KUKA KRL program: ps_ltc_geo_c1_bolha.src, ps_ltc_geo_c1_bolha.dat

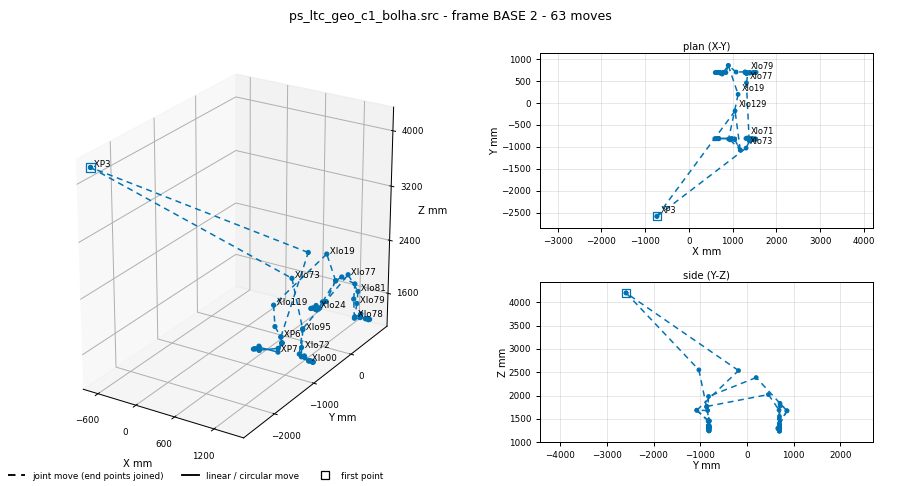
[picture p0: tool path of ps_ltc_geo_c1_bolha.src in frame BASE 2, 63 of 63 moves have a stored position in this frame; points joined in program order, loops and branches not executed]
--- ps_ltc_geo_c1_bolha.src ---
&ACCESS RVO1
&REL 30
&COMMENT SOLDA GEO C1 ACCELO
&PARAM DISKPATH = KRC:\R1\Program\SOLDA LTC
DEF ps_ltc_geo_c1_bolha( )
;FOLD INI
;FOLD SPOTTECH INI

;ENDFOLD (SPOTTECH INI)
;FOLD GRIPPERTECH INI
USER_GRP(0,DUMMY,DUMMY,GDEFAULT)
;ENDFOLD (GRIPPERTECH INI)
  ;FOLD USER INI
    ;Make your modifications here

  ;ENDFOLD (USER INI)
;ENDFOLD (INI)

; Caracterização dos meios de produção:
; Versão Atual:
; 15/07/2013 12:00 Name: P13.050-R5 CHANGES: Solda Geometria Accelo
; C1

chk_w1_wechs_ok ( )      ; CHECK FERRAMENTA: C1

;FOLD PTP P3 CONT Vel=100 % PDAT34 Tool[1]:Gun C1 Base[2]:ACCELO;%{PE}%R 8.2.20,%MKUKATPBASIS,%CMOVE,%VPTP,%P 1:PTP, 2:P3, 3:C_DIS, 5:100, 7:PDAT34
$BWDSTART=FALSE
PDAT_ACT=PPDAT34
FDAT_ACT=FP3
BAS(#PTP_PARAMS,100)
PTP XP3 C_DIS
;ENDFOLD

if MaxStandMenge (1) then
 MaxStandmengeErreicht (1)
endif

IF (NOT(GHOST())) THEN
if Elektrodenwechsel (1) then
 e_fraes1 ()
endif
ENDIF
;FOLD  ;%{PE}%R 8.2.20,%MKUKATPBASIS,%CCOMMENT,%VNORMAL,%P 2:
;ENDFOLD
;FOLD OUT 3339 'R5 aguarda lib soldar geometria' State=TRUE ;%{PE}%R 8.2.20,%MKUKATPBASIS,%COUT,%VOUTX,%P 2:3339, 3:R5 aguarda lib soldar geometria, 5:TRUE, 6:
$OUT[3339]=TRUE
;ENDFOLD
;FOLD WAIT FOR ( IN 3339 'Aguarda lib soldar geometria' );%{PE}%R 8.2.20,%MKUKATPBASIS,%CEXT_WAIT_FOR,%VEXT_WAIT_FOR,%P 2:, 4:, 5:$IN, 6:3339, 7:Aguarda lib soldar geometria, 9:
WAIT FOR  ( $IN[3339] )
;ENDFOLD
;FOLD OUT 3339 'R5 aguarda lib soldar geometria' State=FALSE ;%{PE}%R 8.2.20,%MKUKATPBASIS,%COUT,%VOUTX,%P 2:3339, 3:R5 aguarda lib soldar geometria, 5:FALSE, 6:
$OUT[3339]=FALSE
;ENDFOLD
;FOLD OUT 3344 'R5 entregou peca geo' State=FALSE ;%{PE}%R 8.2.20,%MKUKATPBASIS,%COUT,%VOUTX,%P 2:3344, 3:R5 entregou peca geo, 5:FALSE, 6:
$OUT[3344]=FALSE
;ENDFOLD

;FOLD PTP lo73 CONT Vel=100 % P_OLP1 Tool[1]:Gun C1 Base[2]:ACCELO;%{PE}%R 8.2.20,%MKUKATPBASIS,%CMOVE,%VPTP,%P 1:PTP, 2:lo73, 3:C_DIS, 5:100, 7:P_OLP1
$BWDSTART=FALSE
PDAT_ACT=PP_OLP1
FDAT_ACT=Flo73
BAS(#PTP_PARAMS,100)
PTP Xlo73 C_DIS
;ENDFOLD


;aqui
;FOLD PTP lo95 CONT Vel=100 % P_OLP10 Tool[1]:Gun C1 Base[2]:ACCELO;%{PE}%R8.2,%MKUKATPBASIS,%CMOVE,%VPTP,%P 1:PTP, 2:lo95, 3:C_DIS, 5:100, 7:P_OLP10
$BWDSTART = FALSE
PDAT_ACT= PP_OLP10
FDAT_ACT= Flo95
BAS(#PTP_PARAMS,100)
PTP Xlo95 C_DIS
;ENDFOLD
;FOLD PTP lo72 CONT Vel=100 % P_OLP11 Tool[1]:Gun C1 Base[2]:ACCELO;%{PE}%R8.2,%MKUKATPBASIS,%CMOVE,%VPTP,%P 1:PTP, 2:lo72, 3:C_DIS, 5:100, 7:P_OLP11
$BWDSTART = FALSE
PDAT_ACT= PP_OLP11
FDAT_ACT= Flo72
BAS(#PTP_PARAMS,100)
PTP Xlo72 C_DIS
;ENDFOLD


;FOLD PTP lo71 CONT Vel=100 % P_OLP12 Tool[1]:Gun C1 Base[2]:ACCELO;%{PE}%R8.2,%MKUKATPBASIS,%CMOVE,%VPTP,%P 1:PTP, 2:lo71, 3:C_DIS, 5:100, 7:P_OLP12
$BWDSTART = FALSE
PDAT_ACT= PP_OLP12
FDAT_ACT= Flo71
BAS(#PTP_PARAMS,100)
PTP Xlo71 C_DIS
;ENDFOLD
;FOLD PTP lo00 CONT Vel=100 % PDAT1 Tool[1]:Gun C1 Base[2]:ACCELO;%{PE}%R 8.2.20,%MKUKATPBASIS,%CMOVE,%VPTP,%P 1:PTP, 2:lo00, 3:C_DIS, 5:100, 7:PDAT1
$BWDSTART=FALSE
PDAT_ACT=PPDAT1
FDAT_ACT=Flo00
BAS(#PTP_PARAMS,100)
PTP Xlo00 C_DIS
;ENDFOLD
;FOLD PTP lo01 CONT Vel=100 % PDAT2 Tool[1]:Gun C1 Base[2]:ACCELO;%{PE}%R 8.2.20,%MKUKATPBASIS,%CMOVE,%VPTP,%P 1:PTP, 2:lo01, 3:C_DIS, 5:100, 7:PDAT2
$BWDSTART=FALSE
PDAT_ACT=PPDAT2
FDAT_ACT=Flo01
BAS(#PTP_PARAMS,100)
PTP Xlo01 C_DIS
;ENDFOLD

;FOLD ; swp_60_0421;%{PE}%R 8.2.20,%MKUKATPBASIS,%CCOMMENT,%VNORMAL,%P 2:swp_60_0421
;ENDFOLD
;FOLD PTP lpt_60_0421 P_OLP13 SPOT Gun=1 RETR CLS PgNo1=2 ACTIVE=1 Tool[1]:Gun C1 Base[2]:ACCELO;%{PE}%R 8.2.2,%MKUKATPSPOT,%CSPOT,%VPTP,%P 1:PTP, 2:lpt_60_0421, 3:, 5:100, 7:P_OLP13, 10:1, 12:#FIRST, 14:#CLO, 16:2, 18:1, 20:1, 22:0, 24:1, 25:S_OLP2
$BWDSTART=FALSE
PDAT_ACT=PP_OLP13
FDAT_ACT=Flpt_60_0421
BAS(#PTP_PARAMS,PP_OLP13.VEL)
S_ACT.GUN=1
S_ACT.PAIR=SDEFAULT.PAIR
S_ACT.RETR=#CLO
S_ACT.CLO_TM=1
S_ACT.PGNO1=2
S_ACT.PGNO2=SDEFAULT.PGNO2
S_ACT.PRESS1=SDEFAULT.PRESS1
S_ACT.PRESS2=SDEFAULT.PRESS2
S_READY=FALSE
PTP Xlpt_60_0421
USERSPOT(#SPOT, S_ACT)
WAIT FOR S_READY
;ENDFOLD

;FOLD ; swp_60_0419;%{PE}%R 8.2.20,%MKUKATPBASIS,%CCOMMENT,%VNORMAL,%P 2:swp_60_0419
;ENDFOLD
;FOLD PTP lpt_60_0419 P_OLP14 SPOT Gun=1 RETR CLS PgNo1=3 ACTIVE=1 Tool[1]:Gun C1 Base[2]:ACCELO;%{PE}%R 8.2.2,%MKUKATPSPOT,%CSPOT,%VPTP,%P 1:PTP, 2:lpt_60_0419, 3:, 5:100, 7:P_OLP14, 10:1, 12:#FIRST, 14:#CLO, 16:3, 18:1, 20:1, 22:0, 24:1, 25:S_OLP3
$BWDSTART=FALSE
PDAT_ACT=PP_OLP14
FDAT_ACT=Flpt_60_0419
BAS(#PTP_PARAMS,PP_OLP14.VEL)
S_ACT.GUN=1
S_ACT.PAIR=SDEFAULT.PAIR
S_ACT.RETR=#CLO
S_ACT.CLO_TM=1
S_ACT.PGNO1=3
S_ACT.PGNO2=SDEFAULT.PGNO2
S_ACT.PRESS1=SDEFAULT.PRESS1
S_ACT.PRESS2=SDEFAULT.PRESS2
S_READY=FALSE
PTP Xlpt_60_0419
USERSPOT(#SPOT, S_ACT)
WAIT FOR S_READY
;ENDFOLD

;FOLD ; swp_60_0417;%{PE}%R 8.2.20,%MKUKATPBASIS,%CCOMMENT,%VNORMAL,%P 2:swp_60_0417
;ENDFOLD
;FOLD PTP lpt_60_0417 P_OLP15 SPOT Gun=1 RETR CLS PgNo1=4 ACTIVE=1 Tool[1]:Gun C1 Base[2]:ACCELO;%{PE}%R 8.2.2,%MKUKATPSPOT,%CSPOT,%VPTP,%P 1:PTP, 2:lpt_60_0417, 3:, 5:100, 7:P_OLP15, 10:1, 12:#FIRST, 14:#CLO, 16:4, 18:1, 20:1, 22:0, 24:1, 25:S_OLP4
$BWDSTART=FALSE
PDAT_ACT=PP_OLP15
FDAT_ACT=Flpt_60_0417
BAS(#PTP_PARAMS,PP_OLP15.VEL)
S_ACT.GUN=1
S_ACT.PAIR=SDEFAULT.PAIR
S_ACT.RETR=#CLO
S_ACT.CLO_TM=1
S_ACT.PGNO1=4
S_ACT.PGNO2=SDEFAULT.PGNO2
S_ACT.PRESS1=SDEFAULT.PRESS1
S_ACT.PRESS2=SDEFAULT.PRESS2
S_READY=FALSE
PTP Xlpt_60_0417
USERSPOT(#SPOT, S_ACT)
WAIT FOR S_READY
;ENDFOLD

;FOLD ; swp_60_0415;%{PE}%R 8.2.20,%MKUKATPBASIS,%CCOMMENT,%VNORMAL,%P 2:swp_60_0415
;ENDFOLD
;FOLD PTP lpt_60_0415 P_OLP16 SPOT Gun=1 RETR OPN PgNo1=5 ACTIVE=1 Tool[1]:Gun C1 Base[2]:ACCELO;%{PE}%R 8.2.2,%MKUKATPSPOT,%CSPOT,%VPTP,%P 1:PTP, 2:lpt_60_0415, 3:, 5:100, 7:P_OLP16, 10:1, 12:#FIRST, 14:#OPN, 16:5, 18:1, 20:1, 22:0, 24:1, 25:S_OLP5
$BWDSTART=FALSE
PDAT_ACT=PP_OLP16
FDAT_ACT=Flpt_60_0415
BAS(#PTP_PARAMS,PP_OLP16.VEL)
S_ACT.GUN=1
S_ACT.PAIR=SDEFAULT.PAIR
S_ACT.RETR=#OPN
S_ACT.CLO_TM=1
S_ACT.PGNO1=5
S_ACT.PGNO2=SDEFAULT.PGNO2
S_ACT.PRESS1=SDEFAULT.PRESS1
S_ACT.PRESS2=SDEFAULT.PRESS2
S_READY=FALSE
PTP Xlpt_60_0415
USERSPOT(#SPOT, S_ACT)
WAIT FOR S_READY
;ENDFOLD

;FOLD PTP lo75 CONT Vel=100 % P_OLP17 Tool[1]:Gun C1 Base[2]:ACCELO;%{PE}%R8.2,%MKUKATPBASIS,%CMOVE,%VPTP,%P 1:PTP, 2:lo75, 3:C_DIS, 5:100, 7:P_OLP17
$BWDSTART = FALSE
PDAT_ACT= PP_OLP17
FDAT_ACT= Flo75
BAS(#PTP_PARAMS,100)
PTP Xlo75 C_DIS
;ENDFOLD

;FOLD ; swp_60_0413;%{PE}%R 8.2.20,%MKUKATPBASIS,%CCOMMENT,%VNORMAL,%P 2:swp_60_0413
;ENDFOLD
;FOLD PTP lpt_60_0413 P_OLP18 SPOT Gun=1 RETR OPN PgNo1=6 ACTIVE=1 Tool[1]:Gun C1 Base[2]:ACCELO;%{PE}%R 8.2.2,%MKUKATPSPOT,%CSPOT,%VPTP,%P 1:PTP, 2:lpt_60_0413, 3:, 5:100, 7:P_OLP18, 10:1, 12:#FIRST, 14:#OPN, 16:6, 18:1, 20:1, 22:0, 24:1, 25:S_OLP6
$BWDSTART=FALSE
PDAT_ACT=PP_OLP18
FDAT_ACT=Flpt_60_0413
BAS(#PTP_PARAMS,PP_OLP18.VEL)
S_ACT.GUN=1
S_ACT.PAIR=SDEFAULT.PAIR
S_ACT.RETR=#OPN
S_ACT.CLO_TM=1
S_ACT.PGNO1=6
S_ACT.PGNO2=SDEFAULT.PGNO2
S_ACT.PRESS1=SDEFAULT.PRESS1
S_ACT.PRESS2=SDEFAULT.PRESS2
S_READY=FALSE
PTP Xlpt_60_0413
USERSPOT(#SPOT, S_ACT)
WAIT FOR S_READY
;ENDFOLD

;FOLD PTP lo76 CONT Vel=100 % P_OLP19 Tool[1]:Gun C1 Base[2]:ACCELO;%{PE}%R8.2,%MKUKATPBASIS,%CMOVE,%VPTP,%P 1:PTP, 2:lo76, 3:C_DIS, 5:100, 7:P_OLP19
$BWDSTART = FALSE
PDAT_ACT= PP_OLP19
FDAT_ACT= Flo76
BAS(#PTP_PARAMS,100)
PTP Xlo76 C_DIS
;ENDFOLD
;FOLD PTP lo80 CONT Vel=100 % P_OLP20 Tool[1]:Gun C1 Base[2]:ACCELO;%{PE}%R8.2,%MKUKATPBASIS,%CMOVE,%VPTP,%P 1:PTP, 2:lo80, 3:C_DIS, 5:100, 7:P_OLP20
$BWDSTART = FALSE
PDAT_ACT= PP_OLP20
FDAT_ACT= Flo80
BAS(#PTP_PARAMS,100)
PTP Xlo80 C_DIS
;ENDFOLD
;FOLD PTP lo77 CONT Vel=100 % P_OLP21 Tool[1]:Gun C1 Base[2]:ACCELO;%{PE}%R8.2,%MKUKATPBASIS,%CMOVE,%VPTP,%P 1:PTP, 2:lo77, 3:C_DIS, 5:100, 7:P_OLP21
$BWDSTART = FALSE
PDAT_ACT= PP_OLP21
FDAT_ACT= Flo77
BAS(#PTP_PARAMS,100)
PTP Xlo77 C_DIS
;ENDFOLD
;FOLD PTP lo81 CONT Vel=100 % P_OLP22 Tool[1]:Gun C1 Base[2]:ACCELO;%{PE}%R8.2,%MKUKATPBASIS,%CMOVE,%VPTP,%P 1:PTP, 2:lo81, 3:C_DIS, 5:100, 7:P_OLP22
$BWDSTART = FALSE
PDAT_ACT= PP_OLP22
FDAT_ACT= Flo81
BAS(#PTP_PARAMS,100)
PTP Xlo81 C_DIS
;ENDFOLD
;FOLD PTP lo79 CONT Vel=100 % P_OLP23 Tool[1]:Gun C1 Base[2]:ACCELO;%{PE}%R8.2,%MKUKATPBASIS,%CMOVE,%VPTP,%P 1:PTP, 2:lo79, 3:C_DIS, 5:100, 7:P_OLP23
$BWDSTART = FALSE
PDAT_ACT= PP_OLP23
FDAT_ACT= Flo79
BAS(#PTP_PARAMS,100)
PTP Xlo79 C_DIS
;ENDFOLD
;FOLD PTP lo78 CONT Vel=100 % P_OLP24 Tool[1]:Gun C1 Base[2]:ACCELO;%{PE}%R8.2,%MKUKATPBASIS,%CMOVE,%VPTP,%P 1:PTP, 2:lo78, 3:C_DIS, 5:100, 7:P_OLP24
$BWDSTART = FALSE
PDAT_ACT= PP_OLP24
FDAT_ACT= Flo78
BAS(#PTP_PARAMS,100)
PTP Xlo78 C_DIS
;ENDFOLD
;FOLD PTP lo03 CONT Vel=100 % PDAT4 Tool[1]:Gun C1 Base[2]:ACCELO;%{PE}%R 8.2.20,%MKUKATPBASIS,%CMOVE,%VPTP,%P 1:PTP, 2:lo03, 3:C_DIS, 5:100, 7:PDAT4
$BWDSTART=FALSE
PDAT_ACT=PPDAT4
FDAT_ACT=Flo03
BAS(#PTP_PARAMS,100)
PTP Xlo03 C_DIS
;ENDFOLD

;FOLD ; swp_60_0414;%{PE}%R 8.2.20,%MKUKATPBASIS,%CCOMMENT,%VNORMAL,%P 2:swp_60_0414
;ENDFOLD
;FOLD PTP lpt_60_0414 P_OLP25 SPOT Gun=1 RETR OPN PgNo1=7 ACTIVE=1 Tool[1]:Gun C1 Base[2]:ACCELO;%{PE}%R 8.2.2,%MKUKATPSPOT,%CSPOT,%VPTP,%P 1:PTP, 2:lpt_60_0414, 3:, 5:100, 7:P_OLP25, 10:1, 12:#FIRST, 14:#OPN, 16:7, 18:1, 20:1, 22:0, 24:1, 25:S_OLP7
$BWDSTART=FALSE
PDAT_ACT=PP_OLP25
FDAT_ACT=Flpt_60_0414
BAS(#PTP_PARAMS,PP_OLP25.VEL)
S_ACT.GUN=1
S_ACT.PAIR=SDEFAULT.PAIR
S_ACT.RETR=#OPN
S_ACT.CLO_TM=1
S_ACT.PGNO1=7
S_ACT.PGNO2=SDEFAULT.PGNO2
S_ACT.PRESS1=SDEFAULT.PRESS1
S_ACT.PRESS2=SDEFAULT.PRESS2
S_READY=FALSE
PTP Xlpt_60_0414
USERSPOT(#SPOT, S_ACT)
WAIT FOR S_READY
;ENDFOLD

;FOLD PTP lo82 CONT Vel=100 % P_OLP26 Tool[1]:Gun C1 Base[2]:ACCELO;%{PE}%R8.2,%MKUKATPBASIS,%CMOVE,%VPTP,%P 1:PTP, 2:lo82, 3:C_DIS, 5:100, 7:P_OLP26
$BWDSTART = FALSE
PDAT_ACT= PP_OLP26
FDAT_ACT= Flo82
BAS(#PTP_PARAMS,100)
PTP Xlo82 C_DIS
;ENDFOLD

;FOLD ; swp_60_0416;%{PE}%R 8.2.20,%MKUKATPBASIS,%CCOMMENT,%VNORMAL,%P 2:swp_60_0416
;ENDFOLD
;FOLD PTP lpt_60_0416 P_OLP27 SPOT Gun=1 RETR CLS PgNo1=8 ACTIVE=1 Tool[1]:Gun C1 Base[2]:ACCELO;%{PE}%R 8.2.2,%MKUKATPSPOT,%CSPOT,%VPTP,%P 1:PTP, 2:lpt_60_0416, 3:, 5:100, 7:P_OLP27, 10:1, 12:#FIRST, 14:#CLO, 16:8, 18:1, 20:1, 22:0, 24:1, 25:S_OLP8
$BWDSTART=FALSE
PDAT_ACT=PP_OLP27
FDAT_ACT=Flpt_60_0416
BAS(#PTP_PARAMS,PP_OLP27.VEL)
S_ACT.GUN=1
S_ACT.PAIR=SDEFAULT.PAIR
S_ACT.RETR=#CLO
S_ACT.CLO_TM=1
S_ACT.PGNO1=8
S_ACT.PGNO2=SDEFAULT.PGNO2
S_ACT.PRESS1=SDEFAULT.PRESS1
S_ACT.PRESS2=SDEFAULT.PRESS2
S_READY=FALSE
PTP Xlpt_60_0416
USERSPOT(#SPOT, S_ACT)
WAIT FOR S_READY
;ENDFOLD

;FOLD ; swp_60_0418;%{PE}%R 8.2.20,%MKUKATPBASIS,%CCOMMENT,%VNORMAL,%P 2:swp_60_0418
;ENDFOLD
;FOLD PTP lpt_60_0418 P_OLP28 SPOT Gun=1 RETR CLS PgNo1=9 ACTIVE=1 Tool[1]:Gun C1 Base[2]:ACCELO;%{PE}%R 8.2.2,%MKUKATPSPOT,%CSPOT,%VPTP,%P 1:PTP, 2:lpt_60_0418, 3:, 5:100, 7:P_OLP28, 10:1, 12:#FIRST, 14:#CLO, 16:9, 18:1, 20:1, 22:0, 24:1, 25:S_OLP9
$BWDSTART=FALSE
PDAT_ACT=PP_OLP28
FDAT_ACT=Flpt_60_0418
BAS(#PTP_PARAMS,PP_OLP28.VEL)
S_ACT.GUN=1
S_ACT.PAIR=SDEFAULT.PAIR
S_ACT.RETR=#CLO
S_ACT.CLO_TM=1
S_ACT.PGNO1=9
S_ACT.PGNO2=SDEFAULT.PGNO2
S_ACT.PRESS1=SDEFAULT.PRESS1
S_ACT.PRESS2=SDEFAULT.PRESS2
S_READY=FALSE
PTP Xlpt_60_0418
USERSPOT(#SPOT, S_ACT)
WAIT FOR S_READY
;ENDFOLD

;FOLD ; swp_60_0420;%{PE}%R 8.2.20,%MKUKATPBASIS,%CCOMMENT,%VNORMAL,%P 2:swp_60_0420
;ENDFOLD
;FOLD PTP lpt_60_0420 P_OLP29 SPOT Gun=1 RETR CLS PgNo1=10 ACTIVE=1 Tool[1]:Gun C1 Base[2]:ACCELO;%{PE}%R 8.2.2,%MKUKATPSPOT,%CSPOT,%VPTP,%P 1:PTP, 2:lpt_60_0420, 3:, 5:100, 7:P_OLP29, 10:1, 12:#FIRST, 14:#CLO, 16:10, 18:1, 20:1, 22:0, 24:1, 25:S_OLP10
$BWDSTART=FALSE
PDAT_ACT=PP_OLP29
FDAT_ACT=Flpt_60_0420
BAS(#PTP_PARAMS,PP_OLP29.VEL)
S_ACT.GUN=1
S_ACT.PAIR=SDEFAULT.PAIR
S_ACT.RETR=#CLO
S_ACT.CLO_TM=1
S_ACT.PGNO1=10
S_ACT.PGNO2=SDEFAULT.PGNO2
S_ACT.PRESS1=SDEFAULT.PRESS1
S_ACT.PRESS2=SDEFAULT.PRESS2
S_READY=FALSE
PTP Xlpt_60_0420
USERSPOT(#SPOT, S_ACT)
WAIT FOR S_READY
;ENDFOLD

;FOLD PTP lo04 CONT Vel=100 % PDAT5 Tool[1]:Gun C1 Base[2]:ACCELO;%{PE}%R 8.2.20,%MKUKATPBASIS,%CMOVE,%VPTP,%P 1:PTP, 2:lo04, 3:C_DIS, 5:100, 7:PDAT5
$BWDSTART=FALSE
PDAT_ACT=PPDAT5
FDAT_ACT=Flo04
BAS(#PTP_PARAMS,100)
PTP Xlo04 C_DIS
;ENDFOLD

;FOLD ; swp_60_0422;%{PE}%R 8.2.20,%MKUKATPBASIS,%CCOMMENT,%VNORMAL,%P 2:swp_60_0422
;ENDFOLD
;FOLD PTP lpt_60_0422 P_OLP30 SPOT Gun=1 RETR OPN PgNo1=11 ACTIVE=1 Tool[1]:Gun C1 Base[2]:ACCELO;%{PE}%R 8.2.2,%MKUKATPSPOT,%CSPOT,%VPTP,%P 1:PTP, 2:lpt_60_0422, 3:, 5:100, 7:P_OLP30, 10:1, 12:#FIRST, 14:#OPN, 16:11, 18:1, 20:1, 22:0, 24:1, 25:S_OLP11
$BWDSTART=FALSE
PDAT_ACT=PP_OLP30
FDAT_ACT=Flpt_60_0422
BAS(#PTP_PARAMS,PP_OLP30.VEL)
S_ACT.GUN=1
S_ACT.PAIR=SDEFAULT.PAIR
S_ACT.RETR=#OPN
S_ACT.CLO_TM=1
S_ACT.PGNO1=11
S_ACT.PGNO2=SDEFAULT.PGNO2
S_ACT.PRESS1=SDEFAULT.PRESS1
S_ACT.PRESS2=SDEFAULT.PRESS2
S_READY=FALSE
PTP Xlpt_60_0422
USERSPOT(#SPOT, S_ACT)
WAIT FOR S_READY
;ENDFOLD

;FOLD PTP lo83 CONT Vel=100 % P_OLP31 Tool[1]:Gun C1 Base[2]:ACCELO;%{PE}%R8.2,%MKUKATPBASIS,%CMOVE,%VPTP,%P 1:PTP, 2:lo83, 3:C_DIS, 5:100, 7:P_OLP31
$BWDSTART = FALSE
PDAT_ACT= PP_OLP31
FDAT_ACT= Flo83
BAS(#PTP_PARAMS,100)
PTP Xlo83 C_DIS
;ENDFOLD
;FOLD PTP lo20 CONT Vel=100 % PDAT18 Tool[1]:Gun C1 Base[2]:ACCELO;%{PE}%R 8.2.20,%MKUKATPBASIS,%CMOVE,%VPTP,%P 1:PTP, 2:lo20, 3:C_DIS, 5:100, 7:PDAT18
$BWDSTART=FALSE
PDAT_ACT=PPDAT18
FDAT_ACT=Flo20
BAS(#PTP_PARAMS,100)
PTP Xlo20 C_DIS
;ENDFOLD
;FOLD PTP lo84 CONT Vel=100 % P_OLP32 Tool[1]:Gun C1 Base[2]:ACCELO;%{PE}%R8.2,%MKUKATPBASIS,%CMOVE,%VPTP,%P 1:PTP, 2:lo84, 3:C_DIS, 5:100, 7:P_OLP32
$BWDSTART = FALSE
PDAT_ACT= PP_OLP32
FDAT_ACT= Flo84
BAS(#PTP_PARAMS,100)
PTP Xlo84 C_DIS
;ENDFOLD
;FOLD PTP lo112 CONT Vel=100 % P_OLP53 Tool[1]:Gun C1 Base[2]:ACCELO;%{PE}%R8.2,%MKUKATPBASIS,%CMOVE,%VPTP,%P 1:PTP, 2:lo112, 3:C_DIS, 5:100, 7:P_OLP53
$BWDSTART = FALSE
PDAT_ACT= PP_OLP53
FDAT_ACT= Flo112
BAS(#PTP_PARAMS,100)
PTP Xlo112 C_DIS
;ENDFOLD
;FOLD PTP lo22 CONT Vel=100 % PDAT25 Tool[1]:Gun C1 Base[2]:ACCELO;%{PE}%R 8.2.20,%MKUKATPBASIS,%CMOVE,%VPTP,%P 1:PTP, 2:lo22, 3:C_DIS, 5:100, 7:PDAT25
$BWDSTART=FALSE
PDAT_ACT=PPDAT25
FDAT_ACT=Flo22
BAS(#PTP_PARAMS,100)
PTP Xlo22 C_DIS
;ENDFOLD
;FOLD PTP lo16 CONT Vel=100 % PDAT15 Tool[1]:Gun C1 Base[2]:ACCELO;%{PE}%R 8.2.20,%MKUKATPBASIS,%CMOVE,%VPTP,%P 1:PTP, 2:lo16, 3:C_DIS, 5:100, 7:PDAT15
$BWDSTART=FALSE
PDAT_ACT=PPDAT15
FDAT_ACT=Flo16
BAS(#PTP_PARAMS,100)
PTP Xlo16 C_DIS
;ENDFOLD
;FOLD PTP lo111 CONT Vel=100 % PDAT21 Tool[1]:Gun C1 Base[2]:ACCELO;%{PE}%R 8.2.20,%MKUKATPBASIS,%CMOVE,%VPTP,%P 1:PTP, 2:lo111, 3:C_DIS, 5:100, 7:PDAT21
$BWDSTART=FALSE
PDAT_ACT=PPDAT21
FDAT_ACT=Flo111
BAS(#PTP_PARAMS,100)
PTP Xlo111 C_DIS
;ENDFOLD
;FOLD PTP lo24 CONT Vel=100 % PDAT28 Tool[1]:Gun C1 Base[2]:ACCELO;%{PE}%R 8.2.20,%MKUKATPBASIS,%CMOVE,%VPTP,%P 1:PTP, 2:lo24, 3:C_DIS, 5:100, 7:PDAT28
$BWDSTART=FALSE
PDAT_ACT=PPDAT28
FDAT_ACT=Flo24
BAS(#PTP_PARAMS,100)
PTP Xlo24 C_DIS
;ENDFOLD

;FOLD ; swp_60_0412;%{PE}%R 8.2.20,%MKUKATPBASIS,%CCOMMENT,%VNORMAL,%P 2:swp_60_0412
;ENDFOLD
;FOLD PTP lpt_60_0412 PDAT27 SPOT Gun=1 RETR OPN PgNo1=15 ACTIVE=1 Tool[1]:Gun C1 Base[2]:ACCELO;%{PE}%R 8.2.2,%MKUKATPSPOT,%CSPOT,%VPTP,%P 1:PTP, 2:lpt_60_0412, 3:, 5:100, 7:PDAT27, 10:1, 12:#FIRST, 14:#OPN, 16:15, 18:1, 20:1, 22:0, 24:1, 25:S_OLP15
$BWDSTART=FALSE
PDAT_ACT=PPDAT27
FDAT_ACT=Flpt_60_0412
BAS(#PTP_PARAMS,PPDAT27.VEL)
S_ACT.GUN=1
S_ACT.PAIR=SDEFAULT.PAIR
S_ACT.RETR=#OPN
S_ACT.CLO_TM=1
S_ACT.PGNO1=15
S_ACT.PGNO2=SDEFAULT.PGNO2
S_ACT.PRESS1=SDEFAULT.PRESS1
S_ACT.PRESS2=SDEFAULT.PRESS2
S_READY=FALSE
PTP Xlpt_60_0412
USERSPOT(#SPOT, S_ACT)
WAIT FOR S_READY
;ENDFOLD

;FOLD PTP lo114 CONT Vel=100 % P_OLP58 Tool[1]:Gun C1 Base[2]:ACCELO;%{PE}%R8.2,%MKUKATPBASIS,%CMOVE,%VPTP,%P 1:PTP, 2:lo114, 3:C_DIS, 5:100, 7:P_OLP58
$BWDSTART = FALSE
PDAT_ACT= PP_OLP58
FDAT_ACT= Flo114
BAS(#PTP_PARAMS,100)
PTP Xlo114 C_DIS
;ENDFOLD

;FOLD ; swp_60_0410;%{PE}%R 8.2.20,%MKUKATPBASIS,%CCOMMENT,%VNORMAL,%P 2:swp_60_0410
;ENDFOLD
;FOLD PTP lpt_60_0410 PDAT29 SPOT Gun=1 RETR CLS PgNo1=16 ACTIVE=1 Tool[1]:Gun C1 Base[2]:ACCELO;%{PE}%R 8.2.2,%MKUKATPSPOT,%CSPOT,%VPTP,%P 1:PTP, 2:lpt_60_0410, 3:, 5:100, 7:PDAT29, 10:1, 12:#FIRST, 14:#CLO, 16:16, 18:1, 20:1, 22:0, 24:1, 25:S_OLP16
$BWDSTART=FALSE
PDAT_ACT=PPDAT29
FDAT_ACT=Flpt_60_0410
BAS(#PTP_PARAMS,PPDAT29.VEL)
S_ACT.GUN=1
S_ACT.PAIR=SDEFAULT.PAIR
S_ACT.RETR=#CLO
S_ACT.CLO_TM=1
S_ACT.PGNO1=16
S_ACT.PGNO2=SDEFAULT.PGNO2
S_ACT.PRESS1=SDEFAULT.PRESS1
S_ACT.PRESS2=SDEFAULT.PRESS2
S_READY=FALSE
PTP Xlpt_60_0410
USERSPOT(#SPOT, S_ACT)
WAIT FOR S_READY
;ENDFOLD

;FOLD ; swp_60_0408;%{PE}%R 8.2.20,%MKUKATPBASIS,%CCOMMENT,%VNORMAL,%P 2:swp_60_0408
;ENDFOLD
;FOLD PTP lpt_60_0408 P_OLP60 SPOT Gun=1 RETR CLS PgNo1=17 ACTIVE=1 Tool[1]:Gun C1 Base[2]:ACCELO;%{PE}%R 8.2.2,%MKUKATPSPOT,%CSPOT,%VPTP,%P 1:PTP, 2:lpt_60_0408, 3:, 5:100, 7:P_OLP60, 10:1, 12:#FIRST, 14:#CLO, 16:17, 18:1, 20:1, 22:0, 24:1, 25:S_OLP17
$BWDSTART=FALSE
PDAT_ACT=PP_OLP60
FDAT_ACT=Flpt_60_0408
BAS(#PTP_PARAMS,PP_OLP60.VEL)
S_ACT.GUN=1
S_ACT.PAIR=SDEFAULT.PAIR
S_ACT.RETR=#CLO
S_ACT.CLO_TM=1
S_ACT.PGNO1=17
S_ACT.PGNO2=SDEFAULT.PGNO2
S_ACT.PRESS1=SDEFAULT.PRESS1
S_ACT.PRESS2=SDEFAULT.PRESS2
S_READY=FALSE
PTP Xlpt_60_0408
USERSPOT(#SPOT, S_ACT)
WAIT FOR S_READY
;ENDFOLD

;FOLD ; swp_60_0406;%{PE}%R 8.2.20,%MKUKATPBASIS,%CCOMMENT,%VNORMAL,%P 2:swp_60_0406
;ENDFOLD
;FOLD PTP lpt_60_0406 P_OLP61 SPOT Gun=1 RETR OPN PgNo1=18 ACTIVE=1 Tool[1]:Gun C1 Base[2]:ACCELO;%{PE}%R 8.2.2,%MKUKATPSPOT,%CSPOT,%VPTP,%P 1:PTP, 2:lpt_60_0406, 3:, 5:100, 7:P_OLP61, 10:1, 12:#FIRST, 14:#OPN, 16:18, 18:1, 20:1, 22:0, 24:1, 25:S_OLP18
$BWDSTART=FALSE
PDAT_ACT=PP_OLP61
FDAT_ACT=Flpt_60_0406
BAS(#PTP_PARAMS,PP_OLP61.VEL)
S_ACT.GUN=1
S_ACT.PAIR=SDEFAULT.PAIR
S_ACT.RETR=#OPN
S_ACT.CLO_TM=1
S_ACT.PGNO1=18
S_ACT.PGNO2=SDEFAULT.PGNO2
S_ACT.PRESS1=SDEFAULT.PRESS1
S_ACT.PRESS2=SDEFAULT.PRESS2
S_READY=FALSE
PTP Xlpt_60_0406
USERSPOT(#SPOT, S_ACT)
WAIT FOR S_READY
;ENDFOLD

;FOLD PTP lo115 CONT Vel=100 % PDAT22 Tool[1]:Gun C1 Base[2]:ACCELO;%{PE}%R 8.2.20,%MKUKATPBASIS,%CMOVE,%VPTP,%P 1:PTP, 2:lo115, 3:C_DIS, 5:100, 7:PDAT22
$BWDSTART=FALSE
PDAT_ACT=PPDAT22
FDAT_ACT=Flo115
BAS(#PTP_PARAMS,100)
PTP Xlo115 C_DIS
;ENDFOLD
;FOLD PTP lo17 CONT Vel=100 % PDAT30 Tool[1]:Gun C1 Base[2]:ACCELO;%{PE}%R 8.2.20,%MKUKATPBASIS,%CMOVE,%VPTP,%P 1:PTP, 2:lo17, 3:C_DIS, 5:100, 7:PDAT30
$BWDSTART=FALSE
PDAT_ACT=PPDAT30
FDAT_ACT=Flo17
BAS(#PTP_PARAMS,100)
PTP Xlo17 C_DIS
;ENDFOLD
;FOLD PTP lo116 CONT Vel=100 % PDAT31 Tool[1]:Gun C1 Base[2]:ACCELO;%{PE}%R 8.2.20,%MKUKATPBASIS,%CMOVE,%VPTP,%P 1:PTP, 2:lo116, 3:C_DIS, 5:100, 7:PDAT31
$BWDSTART=FALSE
PDAT_ACT=PPDAT31
FDAT_ACT=Flo116
BAS(#PTP_PARAMS,100)
PTP Xlo116 C_DIS
;ENDFOLD
;FOLD PTP lo19 CONT Vel=100 % PDAT17 Tool[1]:Gun C1 Base[2]:ACCELO;%{PE}%R 8.2.20,%MKUKATPBASIS,%CMOVE,%VPTP,%P 1:PTP, 2:lo19, 3:C_DIS, 5:100, 7:PDAT17
$BWDSTART=FALSE
PDAT_ACT=PPDAT17
FDAT_ACT=Flo19
BAS(#PTP_PARAMS,100)
PTP Xlo19 C_DIS
;ENDFOLD
;FOLD PTP lo119 CONT Vel=100 % P_OLP66 Tool[1]:Gun C1 Base[2]:ACCELO;%{PE}%R8.2,%MKUKATPBASIS,%CMOVE,%VPTP,%P 1:PTP, 2:lo119, 3:C_DIS, 5:100, 7:P_OLP66
$BWDSTART = FALSE
PDAT_ACT= PP_OLP66
FDAT_ACT= Flo119
BAS(#PTP_PARAMS,100)
PTP Xlo119 C_DIS
;ENDFOLD
;FOLD PTP lo07 CONT Vel=100 % PDAT8 Tool[1]:Gun C1 Base[2]:ACCELO;%{PE}%R 8.2.20,%MKUKATPBASIS,%CMOVE,%VPTP,%P 1:PTP, 2:lo07, 3:C_DIS, 5:100, 7:PDAT8
$BWDSTART=FALSE
PDAT_ACT=PPDAT8
FDAT_ACT=Flo07
BAS(#PTP_PARAMS,100)
PTP Xlo07 C_DIS
;ENDFOLD
;FOLD PTP P6 CONT Vel=100 % PDAT37 Tool[1]:Gun C1 Base[2]:ACCELO;%{PE}%R 8.2.20,%MKUKATPBASIS,%CMOVE,%VPTP,%P 1:PTP, 2:P6, 3:C_DIS, 5:100, 7:PDAT37
$BWDSTART=FALSE
PDAT_ACT=PPDAT37
FDAT_ACT=FP6
BAS(#PTP_PARAMS,100)
PTP XP6 C_DIS
;ENDFOLD
;FOLD PTP P5 CONT Vel=100 % PDAT36 Tool[1]:Gun C1 Base[2]:ACCELO;%{PE}%R 8.2.20,%MKUKATPBASIS,%CMOVE,%VPTP,%P 1:PTP, 2:P5, 3:C_DIS, 5:100, 7:PDAT36
$BWDSTART=FALSE
PDAT_ACT=PPDAT36
FDAT_ACT=FP5
BAS(#PTP_PARAMS,100)
PTP XP5 C_DIS
;ENDFOLD

;FOLD LIN P5 Vel=2 m/s CPDAT25 Tool[1]:Gun C1 Base[2]:ACCELO;%{PE}%R 8.2.20,%MKUKATPBASIS,%CMOVE,%VLIN,%P 1:LIN, 2:P5, 3:, 5:2, 7:CPDAT25
$BWDSTART=FALSE
LDAT_ACT=LCPDAT25
FDAT_ACT=FP5
BAS(#CP_PARAMS,2)
LIN XP5
;ENDFOLD
;FOLD LIN P7 CONT Vel=2 m/s CPDAT26 Tool[1]:Gun C1 Base[2]:ACCELO;%{PE}%R 8.2.20,%MKUKATPBASIS,%CMOVE,%VLIN,%P 1:LIN, 2:P7, 3:C_DIS C_DIS, 5:2, 7:CPDAT26
$BWDSTART=FALSE
LDAT_ACT=LCPDAT26
FDAT_ACT=FP7
BAS(#CP_PARAMS,2)
LIN XP7 C_DIS C_DIS
;ENDFOLD
;FOLD LIN lo124 CONT Vel=0.5 m/s CPDAT4 Tool[1]:Gun C1 Base[2]:ACCELO;%{PE}%R 8.2.20,%MKUKATPBASIS,%CMOVE,%VLIN,%P 1:LIN, 2:lo124, 3:C_DIS C_DIS, 5:0.5, 7:CPDAT4
$BWDSTART=FALSE
LDAT_ACT=LCPDAT4
FDAT_ACT=Flo124
BAS(#CP_PARAMS,0.5)
LIN Xlo124 C_DIS C_DIS
;ENDFOLD

;FOLD ; swp_60_0411;%{PE}%R 8.2.20,%MKUKATPBASIS,%CCOMMENT,%VNORMAL,%P 2:swp_60_0411
;ENDFOLD
;FOLD PTP lpt_60_0411 P_OLP71 SPOT Gun=1 RETR OPN PgNo1=19 ACTIVE=1 Tool[1]:Gun C1 Base[2]:ACCELO;%{PE}%R 8.2.2,%MKUKATPSPOT,%CSPOT,%VPTP,%P 1:PTP, 2:lpt_60_0411, 3:, 5:100, 7:P_OLP71, 10:1, 12:#FIRST, 14:#OPN, 16:19, 18:1, 20:1, 22:0, 24:1, 25:S_OLP19
$BWDSTART=FALSE
PDAT_ACT=PP_OLP71
FDAT_ACT=Flpt_60_0411
BAS(#PTP_PARAMS,PP_OLP71.VEL)
S_ACT.GUN=1
S_ACT.PAIR=SDEFAULT.PAIR
S_ACT.RETR=#OPN
S_ACT.CLO_TM=1
S_ACT.PGNO1=19
S_ACT.PGNO2=SDEFAULT.PGNO2
S_ACT.PRESS1=SDEFAULT.PRESS1
S_ACT.PRESS2=SDEFAULT.PRESS2
S_READY=FALSE
PTP Xlpt_60_0411
USERSPOT(#SPOT, S_ACT)
WAIT FOR S_READY
;ENDFOLD

;FOLD LIN lo125 CONT Vel=0.5 m/s CPDAT6 Tool[1]:Gun C1 Base[2]:ACCELO;%{PE}%R 8.2.20,%MKUKATPBASIS,%CMOVE,%VLIN,%P 1:LIN, 2:lo125, 3:C_DIS C_DIS, 5:0.5, 7:CPDAT6
$BWDSTART=FALSE
LDAT_ACT=LCPDAT6
FDAT_ACT=Flo125
BAS(#CP_PARAMS,0.5)
LIN Xlo125 C_DIS C_DIS
;ENDFOLD

;FOLD ; swp_60_0409;%{PE}%R 8.2.20,%MKUKATPBASIS,%CCOMMENT,%VNORMAL,%P 2:swp_60_0409
;ENDFOLD
;FOLD LIN lpt_60_0409 CPDAT11 SPOT Gun=1 RETR CLS PgNo1=20 ACTIVE=1 Tool[1]:Gun C1 Base[2]:ACCELO;%{PE}%R 8.2.2,%MKUKATPSPOT,%CSPOT,%VLIN,%P 1:LIN, 2:lpt_60_0409, 3:, 5:2, 7:CPDAT11, 10:1, 12:#FIRST, 14:#CLO, 16:20, 18:1, 20:1, 22:0, 24:1, 25:S_OLP20
$BWDSTART=FALSE
LDAT_ACT=LCPDAT11
FDAT_ACT=Flpt_60_0409
BAS(#CP_PARAMS,LCPDAT11.VEL)
S_ACT.GUN=1
S_ACT.PAIR=SDEFAULT.PAIR
S_ACT.RETR=#CLO
S_ACT.CLO_TM=1
S_ACT.PGNO1=20
S_ACT.PGNO2=SDEFAULT.PGNO2
S_ACT.PRESS1=SDEFAULT.PRESS1
S_ACT.PRESS2=SDEFAULT.PRESS2
S_READY=FALSE
LIN Xlpt_60_0409
USERSPOT(#SPOT, S_ACT)
WAIT FOR S_READY
;ENDFOLD

;FOLD ; swp_60_0407;%{PE}%R 8.2.20,%MKUKATPBASIS,%CCOMMENT,%VNORMAL,%P 2:swp_60_0407
;ENDFOLD
;FOLD LIN lpt_60_0407 CPDAT12 SPOT Gun=1 RETR CLS PgNo1=21 ACTIVE=1 Tool[1]:Gun C1 Base[2]:ACCELO;%{PE}%R 8.2.2,%MKUKATPSPOT,%CSPOT,%VLIN,%P 1:LIN, 2:lpt_60_0407, 3:, 5:2, 7:CPDAT12, 10:1, 12:#FIRST, 14:#CLO, 16:21, 18:1, 20:1, 22:0, 24:1, 25:S_OLP21
$BWDSTART=FALSE
LDAT_ACT=LCPDAT12
FDAT_ACT=Flpt_60_0407
BAS(#CP_PARAMS,LCPDAT12.VEL)
S_ACT.GUN=1
S_ACT.PAIR=SDEFAULT.PAIR
S_ACT.RETR=#CLO
S_ACT.CLO_TM=1
S_ACT.PGNO1=21
S_ACT.PGNO2=SDEFAULT.PGNO2
S_ACT.PRESS1=SDEFAULT.PRESS1
S_ACT.PRESS2=SDEFAULT.PRESS2
S_READY=FALSE
LIN Xlpt_60_0407
USERSPOT(#SPOT, S_ACT)
WAIT FOR S_READY
;ENDFOLD

;FOLD ; swp_60_0405;%{PE}%R 8.2.20,%MKUKATPBASIS,%CCOMMENT,%VNORMAL,%P 2:swp_60_0405
;ENDFOLD
;FOLD LIN lpt_60_0405 CPDAT13 SPOT Gun=1 RETR OPN PgNo1=22 ACTIVE=1 Tool[1]:Gun C1 Base[2]:ACCELO;%{PE}%R 8.2.2,%MKUKATPSPOT,%CSPOT,%VLIN,%P 1:LIN, 2:lpt_60_0405, 3:, 5:2, 7:CPDAT13, 10:1, 12:#FIRST, 14:#OPN, 16:22, 18:1, 20:1, 22:0, 24:1, 25:S_OLP22
$BWDSTART=FALSE
LDAT_ACT=LCPDAT13
FDAT_ACT=Flpt_60_0405
BAS(#CP_PARAMS,LCPDAT13.VEL)
S_ACT.GUN=1
S_ACT.PAIR=SDEFAULT.PAIR
S_ACT.RETR=#OPN
S_ACT.CLO_TM=1
S_ACT.PGNO1=22
S_ACT.PGNO2=SDEFAULT.PGNO2
S_ACT.PRESS1=SDEFAULT.PRESS1
S_ACT.PRESS2=SDEFAULT.PRESS2
S_READY=FALSE
LIN Xlpt_60_0405
USERSPOT(#SPOT, S_ACT)
WAIT FOR S_READY
;ENDFOLD

;FOLD LIN lo126 CONT Vel=0.1 m/s CPDAT14 Tool[1]:Gun C1 Base[2]:ACCELO;%{PE}%R 8.2.20,%MKUKATPBASIS,%CMOVE,%VLIN,%P 1:LIN, 2:lo126, 3:C_DIS C_DIS, 5:0.1, 7:CPDAT14
$BWDSTART=FALSE
LDAT_ACT=LCPDAT14
FDAT_ACT=Flo126
BAS(#CP_PARAMS,0.1)
LIN Xlo126 C_DIS C_DIS
;ENDFOLD
;FOLD LIN lo127 CONT Vel=2 m/s CPDAT15 Tool[1]:Gun C1 Base[2]:ACCELO;%{PE}%R 8.2.20,%MKUKATPBASIS,%CMOVE,%VLIN,%P 1:LIN, 2:lo127, 3:C_DIS C_DIS, 5:2, 7:CPDAT15
$BWDSTART=FALSE
LDAT_ACT=LCPDAT15
FDAT_ACT=Flo127
BAS(#CP_PARAMS,2)
LIN Xlo127 C_DIS C_DIS
;ENDFOLD
;FOLD LIN lo128 CONT Vel=2 m/s CPDAT16 Tool[1]:Gun C1 Base[2]:ACCELO;%{PE}%R 8.2.20,%MKUKATPBASIS,%CMOVE,%VLIN,%P 1:LIN, 2:lo128, 3:C_DIS C_DIS, 5:2, 7:CPDAT16
$BWDSTART=FALSE
LDAT_ACT=LCPDAT16
FDAT_ACT=Flo128
BAS(#CP_PARAMS,2)
LIN Xlo128 C_DIS C_DIS
;ENDFOLD

;FOLD PTP P8 Vel=100 % PDAT39 Tool[1]:Gun C1 Base[2]:ACCELO;%{PE}%R 8.2.20,%MKUKATPBASIS,%CMOVE,%VPTP,%P 1:PTP, 2:P8, 3:, 5:100, 7:PDAT39
$BWDSTART=FALSE
PDAT_ACT=PPDAT39
FDAT_ACT=FP8
BAS(#PTP_PARAMS,100)
PTP XP8
;ENDFOLD
;FOLD PTP P9 Vel=100 % PDAT40 Tool[1]:Gun C1 Base[2]:ACCELO;%{PE}%R 8.2.20,%MKUKATPBASIS,%CMOVE,%VPTP,%P 1:PTP, 2:P9, 3:, 5:100, 7:PDAT40
$BWDSTART=FALSE
PDAT_ACT=PPDAT40
FDAT_ACT=FP9
BAS(#PTP_PARAMS,100)
PTP XP9
;ENDFOLD
;FOLD PTP lo129 CONT Vel=50 % P_OLP79 Tool[1]:Gun C1 Base[2]:ACCELO;%{PE}%R 8.2.20,%MKUKATPBASIS,%CMOVE,%VPTP,%P 1:PTP, 2:lo129, 3:C_DIS, 5:50, 7:P_OLP79
$BWDSTART=FALSE
PDAT_ACT=PP_OLP79
FDAT_ACT=Flo129
BAS(#PTP_PARAMS,50)
PTP Xlo129 C_DIS
;ENDFOLD

IF (NOT(GHOST())) THEN
if FraesAnf (1) then
f_fraes1 ()
endif
ENDIF

;FOLD PTP P4 CONT Vel=100 % PDAT35 Tool[1]:Gun C1 Base[2]:ACCELO;%{PE}%R 8.2.20,%MKUKATPBASIS,%CMOVE,%VPTP,%P 1:PTP, 2:P4, 3:C_DIS, 5:100, 7:PDAT35
$BWDSTART=FALSE
PDAT_ACT=PPDAT35
FDAT_ACT=FP4
BAS(#PTP_PARAMS,100)
PTP XP4 C_DIS
;ENDFOLD

;FOLD OUT 3348 'Fora area GEOBOX' State=TRUE ;%{PE}%R 8.2.20,%MKUKATPBASIS,%COUT,%VOUTX,%P 2:3348, 3:Fora area GEOBOX, 5:TRUE, 6:
$OUT[3348]=TRUE
;ENDFOLD

END

--- ps_ltc_geo_c1_bolha.dat ---
&ACCESS RVO1
&REL 30
&COMMENT SOLDA GEO C1 ACCELO
&PARAM DISKPATH = KRC:\R1\Program\SOLDA LTC
DEFDAT  ps_ltc_geo_c1_bolha
;FOLD EXTERNAL DECLARATIONS;%{PE}%MKUKATPBASIS,%CEXT,%VCOMMON,%P
;FOLD GRIPPERTECH EXT
EXT  H50 (INT  :IN,INT  :IN,INT  :IN,GRP_TYP  :IN )
;ENDFOLD (GRIPPERTECH EXT)
;FOLD SPOTTECH EXT
EXT  USERSPOT (S_COMMAND  :IN,SPOT_TYPE  :IN )
;ENDFOLD (SPOTTECH EXT)
;FOLD BASISTECH EXT;%{PE}%MKUKATPBASIS,%CEXT,%VEXT,%P
EXT  BAS (BAS_COMMAND  :IN,REAL  :IN )
DECL INT SUCCESS
;ENDFOLD (BASISTECH EXT)
;FOLD USER EXT;%{E}%MKUKATPUSER,%CEXT,%VEXT,%P
;Make your modifications here

;ENDFOLD (USER EXT)
;ENDFOLD (EXTERNAL DECLARATIONS)

;# ============ START PATH : swp_p13050r5_ltc_geo_c1 =============
DECL FDAT Flo73={TOOL_NO 1,BASE_NO 2,IPO_FRAME #BASE,POINT2[] " ",TQ_STATE FALSE}
DECL PDAT PP_OLP1={VEL 100.0,ACC 100.0,APO_DIST 0.0,APO_MODE #CDIS}
DECL E6POS Xlo73={X 1307.26697,Y -1027.90295,Z 2549.3479,A -176.886993,B 11.3868504,C -1.95086205,S 2,T 10,E1 0.0,E2 0.0,E3 0.0,E4 0.0,E5 0.0,E6 0.0}
DECL FDAT Flo74={TOOL_NO 1,BASE_NO 2,IPO_FRAME #BASE,POINT2[] " "}
DECL PDAT PP_OLP2={VEL 100.0,ACC 100.0,APO_DIST 100.0,APO_MODE #CDIS}
DECL E6POS Xlo74={X 1360.40503,Y -843.128479,Z 1807.83301,A 137.973999,B 1.45918298,C -3.36514497,S 2,T 10,E1 0.0,E2 0.0,E3 0.0,E4 0.0,E5 0.0,E6 0.0}
DECL FDAT Flo91={TOOL_NO 1,BASE_NO 2,IPO_FRAME #BASE,POINT2[] " "}
DECL PDAT PP_OLP4={VEL 100.0,ACC 100.0,APO_DIST 100.0,APO_MODE #CDIS}
DECL E6POS Xlo91={X 1556.91394,Y -845.981506,Z 1452.25,A 103.756897,B -0.868657827,C -12.6080704,S 2,T 42,E1 0.0,E2 0.0,E3 0.0,E4 0.0,E5 0.0,E6 0.0}
DECL FDAT Flo92={TOOL_NO 1,BASE_NO 2,IPO_FRAME #BASE,POINT2[] " "}
DECL PDAT PP_OLP5={VEL 100.0,ACC 100.0,APO_DIST 100.0,APO_MODE #CDIS}
DECL E6POS Xlo92={X 1591.71204,Y -853.740417,Z 1309.13501,A 103.756798,B -0.868668079,C -12.6080704,S 2,T 42,E1 0.0,E2 0.0,E3 0.0,E4 0.0,E5 0.0,E6 0.0}
DECL FDAT Flpt_60_0945={TOOL_NO 1,BASE_NO 2,IPO_FRAME #BASE,POINT2[] " "}
DECL PDAT PP_OLP7={VEL 100.0,ACC 100.0,APO_DIST 0.0}
DECL SPOT_TYPE SS_OLP1={GUN 1,PAIR #FIRST,RETR #OPN,CLO_TM 0,PGNO1 1,PRESS1 1.0,PGNO2 0,PRESS2 0.0}
DECL E6POS Xlpt_60_0945={X 1567.20398,Y -759.725525,Z 1318.41394,A 108.932098,B -0.151382193,C -6.52496719,S 2,T 42,E1 0.0,E2 0.0,E3 0.0,E4 0.0,E5 0.0,E6 0.0}
DECL FDAT Flo93={TOOL_NO 1,BASE_NO 2,IPO_FRAME #BASE,POINT2[] " "}
DECL PDAT PP_OLP8={VEL 100.0,ACC 100.0,APO_DIST 100.0,APO_MODE #CDIS}
DECL E6POS Xlo93={X 1589.98706,Y -766.398071,Z 1317.82605,A 108.861099,B 0.701730728,C -10.6068001,S 2,T 42,E1 0.0,E2 0.0,E3 0.0,E4 0.0,E5 0.0,E6 0.0}
DECL FDAT Flo94={TOOL_NO 1,BASE_NO 2,IPO_FRAME #BASE,POINT2[] " "}
DECL PDAT PP_OLP9={VEL 100.0,ACC 100.0,APO_DIST 100.0,APO_MODE #CDIS}
DECL E6POS Xlo94={X 1514.46704,Y -786.665283,Z 1733.90295,A 108.860901,B 0.697265387,C -10.6027002,S 2,T 42,E1 0.0,E2 0.0,E3 0.0,E4 0.0,E5 0.0,E6 0.0}
DECL FDAT Flo95={TOOL_NO 1,BASE_NO 2,IPO_FRAME #BASE,POINT2[] " "}
DECL PDAT PP_OLP10={VEL 100.0,ACC 100.0,APO_DIST 100.0,APO_MODE #CDIS}
DECL E6POS Xlo95={X 1385.19604,Y -864.172302,Z 1758.52502,A -0.0216164608,B 0.858044326,C 2.81417489,S 2,T 42,E1 0.0,E2 0.0,E3 0.0,E4 0.0,E5 0.0,E6 0.0}
DECL FDAT Flo72={TOOL_NO 1,BASE_NO 2,IPO_FRAME #BASE,POINT2[] " "}
DECL PDAT PP_OLP11={VEL 100.0,ACC 100.0,APO_DIST 100.0,APO_MODE #CDIS}
DECL E6POS Xlo72={X 1332.73401,Y -800.376587,Z 1455.86401,A -0.127529204,B 0.859506786,C 2.81138611,S 2,T 42,E1 0.0,E2 0.0,E3 0.0,E4 0.0,E5 0.0,E6 0.0}
DECL FDAT Flo71={TOOL_NO 1,BASE_NO 2,IPO_FRAME #BASE,POINT2[] " "}
DECL PDAT PP_OLP12={VEL 100.0,ACC 100.0,APO_DIST 100.0,APO_MODE #CDIS}
DECL E6POS Xlo71={X 1331.00598,Y -799.101318,Z 1317.03296,A -0.1227533,B 0.841355979,C -0.772923708,S 2,T 34,E1 0.0,E2 0.0,E3 0.0,E4 0.0,E5 0.0,E6 0.0}
DECL FDAT Flpt_60_0421={TOOL_NO 1,BASE_NO 2,IPO_FRAME #BASE,POINT2[] " "}
DECL PDAT PP_OLP13={VEL 100.0,ACC 100.0,APO_DIST 0.0}
DECL SPOT_TYPE SS_OLP2={GUN 1,PAIR #FIRST,RETR #OPN,CLO_TM 0,PGNO1 1,PRESS1 1.0,PGNO2 0,PRESS2 0.0}
DECL E6POS Xlpt_60_0421={X 1530.08606,Y -825.711487,Z 1306.47095,A -2.648983,B -2.53605509,C -0.648614585,S 2,T 42,E1 0.0,E2 0.0,E3 0.0,E4 0.0,E5 0.0,E6 0.0}
DECL FDAT Flpt_60_0419={TOOL_NO 1,BASE_NO 2,IPO_FRAME #BASE,POINT2[] " "}
DECL PDAT PP_OLP14={VEL 100.0,ACC 100.0,APO_DIST 0.0}
DECL SPOT_TYPE SS_OLP3={GUN 1,PAIR #FIRST,RETR #OPN,CLO_TM 0,PGNO1 1,PRESS1 1.0,PGNO2 0,PRESS2 0.0}
DECL E6POS Xlpt_60_0419={X 1498.67896,Y -825.210693,Z 1309.36499,A -4.16636515,B -2.86667395,C -0.705857098,S 2,T 42,E1 0.0,E2 0.0,E3 0.0,E4 0.0,E5 0.0,E6 0.0}
DECL FDAT Flpt_60_0417={TOOL_NO 1,BASE_NO 2,IPO_FRAME #BASE,POINT2[] " "}
DECL PDAT PP_OLP15={VEL 100.0,ACC 100.0,APO_DIST 0.0}
DECL SPOT_TYPE SS_OLP4={GUN 1,PAIR #FIRST,RETR #OPN,CLO_TM 0,PGNO1 1,PRESS1 1.0,PGNO2 0,PRESS2 0.0}
DECL E6POS Xlpt_60_0417={X 1479.22205,Y -825.017029,Z 1307.31995,A -4.22205496,B 0.686772585,C -0.636554599,S 2,T 34,E1 0.0,E2 0.0,E3 0.0,E4 0.0,E5 0.0,E6 0.0}
DECL FDAT Flpt_60_0415={TOOL_NO 1,BASE_NO 2,IPO_FRAME #BASE,POINT2[] " "}
DECL PDAT PP_OLP16={VEL 100.0,ACC 100.0,APO_DIST 0.0}
DECL SPOT_TYPE SS_OLP5={GUN 1,PAIR #FIRST,RETR #OPN,CLO_TM 0,PGNO1 1,PRESS1 1.0,PGNO2 0,PRESS2 0.0}
DECL E6POS Xlpt_60_0415={X 1463.30603,Y -825.255188,Z 1306.07397,A -5.22370005,B 1.29011095,C 1.68314803,S 2,T 42,E1 0.0,E2 0.0,E3 0.0,E4 0.0,E5 0.0,E6 0.0}
DECL FDAT Flo75={TOOL_NO 1,BASE_NO 2,IPO_FRAME #BASE,POINT2[] " "}
DECL PDAT PP_OLP17={VEL 100.0,ACC 100.0,APO_DIST 100.0,APO_MODE #CDIS}
DECL E6POS Xlo75={X 1388.72205,Y -806.9422,Z 1323.26501,A -2.93125391,B 4.69280481,C 1.70935798,S 2,T 42,E1 0.0,E2 0.0,E3 0.0,E4 0.0,E5 0.0,E6 0.0}
DECL FDAT Flpt_60_0413={TOOL_NO 1,BASE_NO 2,IPO_FRAME #BASE,POINT2[] " "}
DECL PDAT PP_OLP18={VEL 100.0,ACC 100.0,APO_DIST 0.0}
DECL SPOT_TYPE SS_OLP6={GUN 1,PAIR #FIRST,RETR #OPN,CLO_TM 0,PGNO1 1,PRESS1 1.0,PGNO2 0,PRESS2 0.0}
DECL E6POS Xlpt_60_0413={X 1392.42896,Y -826.823608,Z 1358.56104,A -4.80079603,B -0.298234791,C 1.69437206,S 2,T 42,E1 0.0,E2 0.0,E3 0.0,E4 0.0,E5 0.0,E6 0.0}
DECL FDAT Flo76={TOOL_NO 1,BASE_NO 2,IPO_FRAME #BASE,POINT2[] " "}
DECL PDAT PP_OLP19={VEL 100.0,ACC 100.0,APO_DIST 100.0,APO_MODE #CDIS}
DECL E6POS Xlo76={X 1303.23706,Y -807.731995,Z 1353.37903,A -2.92550397,B 4.6937418,C 1.70903599,S 2,T 34,E1 0.0,E2 0.0,E3 0.0,E4 0.0,E5 0.0,E6 0.0}
DECL FDAT Flo80={TOOL_NO 1,BASE_NO 2,IPO_FRAME #BASE,POINT2[] " "}
DECL PDAT PP_OLP20={VEL 100.0,ACC 100.0,APO_DIST 100.0,APO_MODE #CDIS}
DECL E6POS Xlo80={X 1377.54895,Y -854.655212,Z 1766.771,A -2.92672801,B 4.78473377,C 1.74334204,S 2,T 34,E1 0.0,E2 0.0,E3 0.0,E4 0.0,E5 0.0,E6 0.0}
DECL FDAT Flo77={TOOL_NO 1,BASE_NO 2,IPO_FRAME #BASE,POINT2[] " "}
DECL PDAT PP_OLP21={VEL 100.0,ACC 100.0,APO_DIST 100.0,APO_MODE #CDIS}
DECL E6POS Xlo77={X 1315.33899,Y 462.358093,Z 2020.94202,A -2.96999192,B 4.70782089,C 1.71052396,S 2,T 43,E1 0.0,E2 0.0,E3 0.0,E4 0.0,E5 0.0,E6 0.0}
DECL FDAT Flo81={TOOL_NO 1,BASE_NO 2,IPO_FRAME #BASE,POINT2[] " "}
DECL PDAT PP_OLP22={VEL 100.0,ACC 100.0,APO_DIST 100.0,APO_MODE #CDIS}
DECL E6POS Xlo81={X 1349.41003,Y 689.98053,Z 1688.12598,A -2.96997499,B 4.70671988,C 1.71161997,S 2,T 43,E1 0.0,E2 0.0,E3 0.0,E4 0.0,E5 0.0,E6 0.0}
DECL FDAT Flo79={TOOL_NO 1,BASE_NO 2,IPO_FRAME #BASE,POINT2[] " "}
DECL PDAT PP_OLP23={VEL 100.0,ACC 100.0,APO_DIST 100.0,APO_MODE #CDIS}
DECL E6POS Xlo79={X 1334.14099,Y 696.479126,Z 1498.79297,A -2.96953702,B 4.70641708,C 1.71205699,S 2,T 43,E1 0.0,E2 0.0,E3 0.0,E4 0.0,E5 0.0,E6 0.0}
DECL FDAT Flo78={TOOL_NO 1,BASE_NO 2,IPO_FRAME #BASE,POINT2[] " "}
DECL PDAT PP_OLP24={VEL 100.0,ACC 100.0,APO_DIST 100.0,APO_MODE #CDIS}
DECL E6POS Xlo78={X 1317.49097,Y 673.067017,Z 1299.76196,A -1.63332295,B 4.66961002,C -3.78181195,S 2,T 35,E1 0.0,E2 0.0,E3 0.0,E4 0.0,E5 0.0,E6 0.0}
DECL FDAT Flpt_60_0414={TOOL_NO 1,BASE_NO 2,IPO_FRAME #BASE,POINT2[] " "}
DECL PDAT PP_OLP25={VEL 100.0,ACC 100.0,APO_DIST 0.0}
DECL SPOT_TYPE SS_OLP7={GUN 1,PAIR #FIRST,RETR #OPN,CLO_TM 0,PGNO1 1,PRESS1 1.0,PGNO2 0,PRESS2 0.0}
DECL E6POS Xlpt_60_0414={X 1397.37,Y 702.041016,Z 1352.94495,A 4.969666,B 4.28683519,C 0.263703108,S 2,T 43,E1 0.0,E2 0.0,E3 0.0,E4 0.0,E5 0.0,E6 0.0}
DECL FDAT Flo82={TOOL_NO 1,BASE_NO 2,IPO_FRAME #BASE,POINT2[] " "}
DECL PDAT PP_OLP26={VEL 100.0,ACC 100.0,APO_DIST 100.0,APO_MODE #CDIS}
DECL E6POS Xlo82={X 1394.69495,Y 687.177429,Z 1301.43103,A 2.99167991,B 4.38599682,C -2.01178002,S 2,T 35,E1 0.0,E2 0.0,E3 0.0,E4 0.0,E5 0.0,E6 0.0}
DECL FDAT Flpt_60_0416={TOOL_NO 1,BASE_NO 2,IPO_FRAME #BASE,POINT2[] " "}
DECL PDAT PP_OLP27={VEL 100.0,ACC 100.0,APO_DIST 0.0}
DECL SPOT_TYPE SS_OLP8={GUN 1,PAIR #FIRST,RETR #OPN,CLO_TM 0,PGNO1 1,PRESS1 1.0,PGNO2 0,PRESS2 0.0}
DECL E6POS Xlpt_60_0416={X 1471.79102,Y 698.12738,Z 1299.09595,A 3.58784699,B -4.78813219,C -4.36529207,S 2,T 35,E1 0.0,E2 0.0,E3 0.0,E4 0.0,E5 0.0,E6 0.0}
DECL FDAT Flpt_60_0418={TOOL_NO 1,BASE_NO 2,IPO_FRAME #BASE,POINT2[] " "}
DECL PDAT PP_OLP28={VEL 100.0,ACC 100.0,APO_DIST 0.0}
DECL SPOT_TYPE SS_OLP9={GUN 1,PAIR #FIRST,RETR #OPN,CLO_TM 0,PGNO1 1,PRESS1 1.0,PGNO2 0,PRESS2 0.0}
DECL E6POS Xlpt_60_0418={X 1488.66394,Y 698.862976,Z 1303.19104,A 3.64804411,B -4.82679176,C -3.60330105,S 2,T 35,E1 0.0,E2 0.0,E3 0.0,E4 0.0,E5 0.0,E6 0.0}
DECL FDAT Flpt_60_0420={TOOL_NO 1,BASE_NO 2,IPO_FRAME #BASE,POINT2[] " "}
DECL PDAT PP_OLP29={VEL 100.0,ACC 100.0,APO_DIST 0.0}
DECL SPOT_TYPE SS_OLP10={GUN 1,PAIR #FIRST,RETR #OPN,CLO_TM 0,PGNO1 1,PRESS1 1.0,PGNO2 0,PRESS2 0.0}
DECL E6POS Xlpt_60_0420={X 1505.33301,Y 699.696716,Z 1304.71802,A 3.64894009,B -4.82587194,C -3.60395288,S 2,T 35,E1 0.0,E2 0.0,E3 0.0,E4 0.0,E5 0.0,E6 0.0}
DECL FDAT Flpt_60_0422={TOOL_NO 1,BASE_NO 2,IPO_FRAME #BASE,POINT2[] " ",TQ_STATE FALSE}
DECL PDAT PP_OLP30={VEL 100.0,ACC 100.0,APO_DIST 0.0}
DECL SPOT_TYPE SS_OLP11={GUN 1,PAIR #FIRST,RETR #OPN,CLO_TM 0,PGNO1 1,PRESS1 1.0,PGNO2 0,PRESS2 0.0}
DECL E6POS Xlpt_60_0422={X 1535.11694,Y 703.160522,Z 1305.15405,A 3.64920402,B -4.8250618,C -3.60408711,S 2,T 35,E1 0.0,E2 0.0,E3 0.0,E4 0.0,E5 0.0,E6 0.0}
DECL FDAT Flo83={TOOL_NO 1,BASE_NO 2,IPO_FRAME #BASE,POINT2[] " "}
DECL PDAT PP_OLP31={VEL 100.0,ACC 100.0,APO_DIST 100.0,APO_MODE #CDIS}
DECL E6POS Xlo83={X 1305.50806,Y 685.914673,Z 1269.64197,A 2.03070092,B -4.75611782,C -3.69395995,S 2,T 35,E1 0.0,E2 0.0,E3 0.0,E4 0.0,E5 0.0,E6 0.0}
DECL FDAT Flo84={TOOL_NO 1,BASE_NO 2,IPO_FRAME #BASE,POINT2[] " "}
DECL PDAT PP_OLP32={VEL 100.0,ACC 100.0,APO_DIST 100.0,APO_MODE #CDIS}
DECL E6POS Xlo84={X 1284.72595,Y 714.565674,Z 1776.51196,A 1.11308205,B -4.97086906,C -3.39348602,S 2,T 35,E1 0.0,E2 0.0,E3 0.0,E4 0.0,E5 0.0,E6 0.0}
DECL FDAT Flo85={TOOL_NO 1,BASE_NO 2,IPO_FRAME #BASE,POINT2[] " "}
DECL PDAT PP_OLP33={VEL 100.0,ACC 100.0,APO_DIST 100.0,APO_MODE #CDIS}
DECL E6POS Xlo85={X 1282.26001,Y 713.434875,Z 1737.76001,A -133.177994,B 0.961597621,C 5.8954339,S 2,T 3,E1 0.0,E2 0.0,E3 0.0,E4 0.0,E5 0.0,E6 0.0}
DECL FDAT Flo87={TOOL_NO 1,BASE_NO 2,IPO_FRAME #BASE,POINT2[] " "}
DECL PDAT PP_OLP34={VEL 100.0,ACC 100.0,APO_DIST 100.0,APO_MODE #CDIS}
DECL E6POS Xlo87={X 1522.01001,Y 784.212219,Z 1428.29395,A -107.616898,B -6.54158688,C 11.3902597,S 2,T 3,E1 0.0,E2 0.0,E3 0.0,E4 0.0,E5 0.0,E6 0.0}
DECL FDAT Flo88={TOOL_NO 1,BASE_NO 2,IPO_FRAME #BASE,POINT2[] " "}
DECL PDAT PP_OLP35={VEL 100.0,ACC 100.0,APO_DIST 100.0,APO_MODE #CDIS}
DECL E6POS Xlo88={X 1578.34204,Y 703.340088,Z 1367.66504,A -107.616997,B -6.54167509,C 11.3902197,S 2,T 3,E1 0.0,E2 0.0,E3 0.0,E4 0.0,E5 0.0,E6 0.0}
DECL FDAT Flo86={TOOL_NO 1,BASE_NO 2,IPO_FRAME #BASE,POINT2[] " "}
DECL PDAT PP_OLP36={VEL 100.0,ACC 100.0,APO_DIST 100.0,APO_MODE #CDIS}
DECL E6POS Xlo86={X 1589.28796,Y 691.552429,Z 1298.60205,A -107.616798,B -6.54184484,C 11.3900499,S 2,T 3,E1 0.0,E2 0.0,E3 0.0,E4 0.0,E5 0.0,E6 0.0}
DECL FDAT Flpt_60_0946={TOOL_NO 1,BASE_NO 2,IPO_FRAME #BASE,POINT2[] " "}
DECL PDAT PP_OLP37={VEL 100.0,ACC 100.0,APO_DIST 0.0}
DECL SPOT_TYPE SS_OLP12={GUN 1,PAIR #FIRST,RETR #OPN,CLO_TM 0,PGNO1 1,PRESS1 1.0,PGNO2 0,PRESS2 0.0}
DECL E6POS Xlpt_60_0946={X 1564.68604,Y 656.073608,Z 1311.81897,A -107.379402,B -2.47623992,C 6.27559614,S 2,T 3,E1 0.0,E2 0.0,E3 0.0,E4 0.0,E5 0.0,E6 0.0}
DECL FDAT Flo96={TOOL_NO 1,BASE_NO 2,IPO_FRAME #BASE,POINT2[] " "}
DECL PDAT PP_OLP38={VEL 100.0,ACC 100.0,APO_DIST 5.0,APO_MODE #CDIS}
DECL E6POS Xlo96={X 1589.29395,Y 691.555786,Z 1298.60803,A -107.616699,B -6.54172897,C 11.3901997,S 2,T 3,E1 0.0,E2 0.0,E3 0.0,E4 0.0,E5 0.0,E6 0.0}
DECL FDAT Flo97={TOOL_NO 1,BASE_NO 2,IPO_FRAME #BASE,POINT2[] " "}
DECL PDAT PP_OLP39={VEL 100.0,ACC 100.0,APO_DIST 100.0,APO_MODE #CDIS}
DECL E6POS Xlo97={X 1578.30896,Y 703.289429,Z 1367.59802,A -107.617798,B -6.54328012,C 11.38869,S 2,T 3,E1 0.0,E2 0.0,E3 0.0,E4 0.0,E5 0.0,E6 0.0}
DECL FDAT Flo98={TOOL_NO 1,BASE_NO 2,IPO_FRAME #BASE,POINT2[] " "}
DECL PDAT PP_OLP40={VEL 100.0,ACC 100.0,APO_DIST 100.0,APO_MODE #CDIS}
DECL E6POS Xlo98={X 1341.026,Y 803.884827,Z 1630.97803,A -107.617798,B -6.54332876,C 11.3886499,S 2,T 3,E1 0.0,E2 0.0,E3 0.0,E4 0.0,E5 0.0,E6 0.0}
DECL FDAT Flo99={TOOL_NO 1,BASE_NO 2,IPO_FRAME #BASE,POINT2[] " "}
DECL PDAT PP_OLP41={VEL 100.0,ACC 100.0,APO_DIST 100.0,APO_MODE #CDIS}
DECL E6POS Xlo99={X 1234.31799,Y -111.230797,Z 1941.677,A -177.138397,B 0.09107472,C 3.76472306,S 2,T 2,E1 0.0,E2 0.0,E3 0.0,E4 0.0,E5 0.0,E6 0.0}
DECL FDAT Flo103={TOOL_NO 1,BASE_NO 2,IPO_FRAME #BASE,POINT2[] " "}
DECL PDAT PP_OLP42={VEL 100.0,ACC 100.0,APO_DIST 100.0,APO_MODE #CDIS}
DECL E6POS Xlo103={X 1652.15698,Y -59.5736313,Z 1327.84399,A -168.195908,B 0.408452809,C -0.579553723,S 2,T 10,E1 0.0,E2 0.0,E3 0.0,E4 0.0,E5 0.0,E6 0.0}
DECL FDAT Flpt_60_0927={TOOL_NO 1,BASE_NO 2,IPO_FRAME #BASE,POINT2[] " "}
DECL PDAT PP_OLP45={VEL 100.0,ACC 100.0,APO_DIST 0.0}
DECL SPOT_TYPE SS_OLP13={GUN 1,PAIR #FIRST,RETR #OPN,CLO_TM 0,PGNO1 1,PRESS1 1.0,PGNO2 0,PRESS2 0.0}
DECL E6POS Xlpt_60_0927={X 1569.10498,Y -208.135803,Z 1342.42297,A -152.506302,B 4.68592978,C 6.09177113,S 2,T 2,E1 0.0,E2 0.0,E3 0.0,E4 0.0,E5 0.0,E6 0.0}
DECL FDAT Flo104={TOOL_NO 1,BASE_NO 2,IPO_FRAME #BASE,POINT2[] " "}
DECL PDAT PP_OLP46={VEL 100.0,ACC 100.0,APO_DIST 100.0,APO_MODE #CDIS}
DECL E6POS Xlo104={X 1587.57104,Y -43.4862404,Z 1333.03406,A -176.489197,B 3.963413,C -2.02570295,S 2,T 10,E1 0.0,E2 0.0,E3 0.0,E4 0.0,E5 0.0,E6 0.0}
DECL FDAT Flpt_60_0928={TOOL_NO 1,BASE_NO 2,IPO_FRAME #BASE,POINT2[] " "}
DECL PDAT PP_OLP49={VEL 100.0,ACC 100.0,APO_DIST 0.0}
DECL SPOT_TYPE SS_OLP14={GUN 1,PAIR #FIRST,RETR #OPN,CLO_TM 0,PGNO1 1,PRESS1 1.0,PGNO2 0,PRESS2 0.0}
DECL E6POS Xlpt_60_0928={X 1576.25806,Y 94.2199707,Z 1341.93701,A 164.506302,B 1.20341396,C -5.34275389,S 2,T 10,E1 0.0,E2 0.0,E3 0.0,E4 0.0,E5 0.0,E6 0.0}
DECL FDAT Flo107={TOOL_NO 1,BASE_NO 2,IPO_FRAME #BASE,POINT2[] " "}
DECL PDAT PP_OLP50={VEL 100.0,ACC 100.0,APO_DIST 100.0,APO_MODE #CDIS}
DECL E6POS Xlo107={X 1652.21899,Y -68.1121597,Z 1327.92798,A -177.152695,B 0.315783203,C -0.635786712,S 2,T 10,E1 0.0,E2 0.0,E3 0.0,E4 0.0,E5 0.0,E6 0.0}
DECL FDAT Flo109={TOOL_NO 1,BASE_NO 2,IPO_FRAME #BASE,POINT2[] " "}
DECL PDAT PP_OLP51={VEL 100.0,ACC 100.0,APO_DIST 100.0,APO_MODE #CDIS}
DECL E6POS Xlo109={X 1651.91394,Y -68.1043167,Z 1497.43799,A -177.152298,B 0.306374311,C -0.636651814,S 2,T 10,E1 0.0,E2 0.0,E3 0.0,E4 0.0,E5 0.0,E6 0.0}
DECL FDAT Flo108={TOOL_NO 1,BASE_NO 2,IPO_FRAME #BASE,POINT2[] " "}
DECL PDAT PP_OLP52={VEL 100.0,ACC 100.0,APO_DIST 100.0,APO_MODE #CDIS}
DECL E6POS Xlo108={X 1234.30298,Y -111.259804,Z 1941.61499,A -177.139603,B 0.0879546404,C 3.76434302,S 2,T 2,E1 0.0,E2 0.0,E3 0.0,E4 0.0,E5 0.0,E6 0.0}
DECL FDAT Flo112={TOOL_NO 1,BASE_NO 2,IPO_FRAME #BASE,POINT2[] " "}
DECL PDAT PP_OLP53={VEL 100.0,ACC 100.0,APO_DIST 100.0,APO_MODE #CDIS}
DECL E6POS Xlo112={X 1079.51794,Y 709.711914,Z 1832.81494,A -178.465302,B 0.0837532282,C 3.76458406,S 2,T 35,E1 0.0,E2 0.0,E3 0.0,E4 0.0,E5 0.0,E6 0.0}
DECL FDAT Flo111={TOOL_NO 1,BASE_NO 2,IPO_FRAME #BASE,POINT2[] " "}
DECL E6POS Xlo111={X 760.786072,Y 663.473389,Z 1295.22705,A -176.690002,B 9.96015835,C 5.92471409,S 6,T 27,E1 0.0,E2 0.0,E3 0.0,E4 0.0,E5 0.0,E6 0.0}
DECL FDAT Flpt_60_0412={TOOL_NO 1,BASE_NO 2,IPO_FRAME #BASE,POINT2[] " ",TQ_STATE FALSE}
DECL SPOT_TYPE SS_OLP15={GUN 1,PAIR #FIRST,RETR #OPN,CLO_TM 0,PGNO1 1,PRESS1 1.0,PGNO2 0,PRESS2 0.0}
DECL E6POS Xlpt_60_0412={X 682.633118,Y 703.819275,Z 1299.65698,A 176.610901,B 3.501405,C 1.17134798,S 6,T 27,E1 0.0,E2 0.0,E3 0.0,E4 0.0,E5 0.0,E6 0.0}
DECL FDAT Flo114={TOOL_NO 1,BASE_NO 2,IPO_FRAME #BASE,POINT2[] " "}
DECL PDAT PP_OLP58={VEL 100.0,ACC 100.0,APO_DIST 100.0,APO_MODE #CDIS}
DECL E6POS Xlo114={X 679.399719,Y 699.390015,Z 1237.13196,A 170.165405,B 6.5201931,C 0.6422925,S 6,T 59,E1 0.0,E2 0.0,E3 0.0,E4 0.0,E5 0.0,E6 0.0}
DECL FDAT Flpt_60_0410={TOOL_NO 1,BASE_NO 2,IPO_FRAME #BASE,POINT2[] " "}
DECL SPOT_TYPE SS_OLP16={GUN 1,PAIR #FIRST,RETR #OPN,CLO_TM 0,PGNO1 1,PRESS1 1.0,PGNO2 0,PRESS2 0.0}
DECL E6POS Xlpt_60_0410={X 637.812622,Y 700.613403,Z 1252.43604,A 175.599899,B 17.1111908,C 2.81216407,S 6,T 59,E1 0.0,E2 0.0,E3 0.0,E4 0.0,E5 0.0,E6 0.0}
DECL FDAT Flpt_60_0408={TOOL_NO 1,BASE_NO 2,IPO_FRAME #BASE,POINT2[] " "}
DECL PDAT PP_OLP60={VEL 100.0,ACC 100.0,APO_DIST 0.0}
DECL SPOT_TYPE SS_OLP17={GUN 1,PAIR #FIRST,RETR #OPN,CLO_TM 0,PGNO1 1,PRESS1 1.0,PGNO2 0,PRESS2 0.0}
DECL E6POS Xlpt_60_0408={X 620.939392,Y 697.085388,Z 1243.30505,A 175.600204,B 17.1112995,C 2.81204891,S 6,T 59,E1 0.0,E2 0.0,E3 0.0,E4 0.0,E5 0.0,E6 0.0}
DECL FDAT Flpt_60_0406={TOOL_NO 1,BASE_NO 2,IPO_FRAME #BASE,POINT2[] " "}
DECL PDAT PP_OLP61={VEL 100.0,ACC 100.0,APO_DIST 0.0}
DECL SPOT_TYPE SS_OLP18={GUN 1,PAIR #FIRST,RETR #OPN,CLO_TM 0,PGNO1 1,PRESS1 1.0,PGNO2 0,PRESS2 0.0}
DECL E6POS Xlpt_60_0406={X 601.838623,Y 697.887817,Z 1235.19702,A 175.599594,B 17.1111603,C 2.81051302,S 6,T 59,E1 0.0,E2 0.0,E3 0.0,E4 0.0,E5 0.0,E6 0.0}
DECL FDAT Flo115={TOOL_NO 1,BASE_NO 2,IPO_FRAME #BASE,POINT2[] " "}
DECL E6POS Xlo115={X 721.052612,Y 698.805481,Z 1254.87097,A 173.380493,B 13.6330204,C 2.18225908,S 6,T 59,E1 0.0,E2 0.0,E3 0.0,E4 0.0,E5 0.0,E6 0.0}
DECL FDAT Flo116={TOOL_NO 1,BASE_NO 2,IPO_FRAME #BASE,POINT2[] " "}
DECL E6POS Xlo116={X 900.839294,Y 858.841919,Z 1672.51099,A -166.765305,B 10.6000099,C -6.8331542,S 2,T 11,E1 0.0,E2 0.0,E3 0.0,E4 0.0,E5 0.0,E6 0.0}
DECL FDAT Flo119={TOOL_NO 1,BASE_NO 2,IPO_FRAME #BASE,POINT2[] " "}
DECL PDAT PP_OLP66={VEL 100.0,ACC 100.0,APO_DIST 100.0,APO_MODE #CDIS}
DECL E6POS Xlo119={X 907.790283,Y -820.668213,Z 1978.79297,A 178.698303,B 2.38668299,C 3.70810509,S 6,T 26,E1 0.0,E2 0.0,E3 0.0,E4 0.0,E5 0.0,E6 0.0}
DECL FDAT Flo124={TOOL_NO 1,BASE_NO 2,IPO_FRAME #BASE,POINT2[] " "}
DECL E6POS Xlo124={X 679.562988,Y -808.091187,Z 1290.06104,A 179.435501,B 11.2678604,C 0.728407383,S 2,T 10,E1 0.0,E2 0.0,E3 0.0,E4 0.0,E5 0.0,E6 0.0}
DECL FDAT Flpt_60_0411={TOOL_NO 1,BASE_NO 2,IPO_FRAME #BASE,POINT2[] " "}
DECL PDAT PP_OLP71={VEL 100.0,ACC 100.0,APO_DIST 0.0}
DECL SPOT_TYPE SS_OLP19={GUN 1,PAIR #FIRST,RETR #OPN,CLO_TM 0,PGNO1 1,PRESS1 1.0,PGNO2 0,PRESS2 0.0}
DECL E6POS Xlpt_60_0411={X 679.56073,Y -816.327087,Z 1309.46594,A -178.835205,B 11.2412596,C 1.065889,S 2,T 10,E1 0.0,E2 0.0,E3 0.0,E4 0.0,E5 0.0,E6 0.0}
DECL FDAT Flo125={TOOL_NO 1,BASE_NO 2,IPO_FRAME #BASE,POINT2[] " "}
DECL E6POS Xlo125={X 679.620422,Y -811.643188,Z 1245.60803,A 179.435501,B 11.2678604,C 0.728423595,S 2,T 10,E1 0.0,E2 0.0,E3 0.0,E4 0.0,E5 0.0,E6 0.0}
DECL FDAT Flpt_60_0409={TOOL_NO 1,BASE_NO 2,IPO_FRAME #BASE,POINT2[] " "}
DECL SPOT_TYPE SS_OLP20={GUN 1,PAIR #FIRST,RETR #OPN,CLO_TM 0,PGNO1 1,PRESS1 1.0,PGNO2 0,PRESS2 0.0}
DECL E6POS Xlpt_60_0409={X 626.213684,Y -814.357178,Z 1256.73596,A -178.989899,B 15.3787603,C 0.650337577,S 2,T 10,E1 0.0,E2 0.0,E3 0.0,E4 0.0,E5 0.0,E6 0.0}
DECL FDAT Flpt_60_0407={TOOL_NO 1,BASE_NO 2,IPO_FRAME #BASE,POINT2[] " "}
DECL SPOT_TYPE SS_OLP21={GUN 1,PAIR #FIRST,RETR #OPN,CLO_TM 0,PGNO1 1,PRESS1 1.0,PGNO2 0,PRESS2 0.0}
DECL E6POS Xlpt_60_0407={X 609.584473,Y -813.861328,Z 1248.78296,A -178.337997,B 15.8933001,C 0.198495403,S 2,T 10,E1 0.0,E2 0.0,E3 0.0,E4 0.0,E5 0.0,E6 0.0}
DECL FDAT Flpt_60_0405={TOOL_NO 1,BASE_NO 2,IPO_FRAME #BASE,POINT2[] " "}
DECL SPOT_TYPE SS_OLP22={GUN 1,PAIR #FIRST,RETR #OPN,CLO_TM 0,PGNO1 1,PRESS1 1.0,PGNO2 0,PRESS2 0.0}
DECL E6POS Xlpt_60_0405={X 591.324402,Y -813.858887,Z 1241.40601,A -178.772903,B 15.8932199,C 0.198405504,S 2,T 10,E1 0.0,E2 0.0,E3 0.0,E4 0.0,E5 0.0,E6 0.0}
DECL FDAT Flo126={TOOL_NO 1,BASE_NO 2,IPO_FRAME #BASE,POINT2[] " "}
DECL E6POS Xlo126={X 679.562073,Y -808.749573,Z 1245.66602,A 179.435593,B 11.2678299,C 0.728420019,S 2,T 10,E1 0.0,E2 0.0,E3 0.0,E4 0.0,E5 0.0,E6 0.0}
DECL FDAT Flo127={TOOL_NO 1,BASE_NO 2,IPO_FRAME #BASE,POINT2[] " "}
DECL E6POS Xlo127={X 975.734985,Y -808.586304,Z 1352.26001,A 179.548203,B 19.8236904,C 0.635828078,S 2,T 10,E1 0.0,E2 0.0,E3 0.0,E4 0.0,E5 0.0,E6 0.0}
DECL FDAT Flo128={TOOL_NO 1,BASE_NO 2,IPO_FRAME #BASE,POINT2[] " "}
DECL E6POS Xlo128={X 1043.36804,Y -827.15863,Z 1455.36206,A -177.824005,B 19.4657307,C 3.5938921,S 2,T 10,E1 0.0,E2 0.0,E3 0.0,E4 0.0,E5 0.0,E6 0.0}
DECL FDAT Flo129={TOOL_NO 1,BASE_NO 2,IPO_FRAME #BASE,POINT2[] " "}
DECL PDAT PP_OLP79={VEL 100.0,ACC 100.0,APO_DIST 100.0,APO_MODE #CDIS}
DECL E6POS Xlo129={X 1054.81396,Y -178.232895,Z 2534.1709,A 172.109406,B -4.29547119,C -7.89952278,S 6,T 26,E1 0.0,E2 0.0,E3 0.0,E4 0.0,E5 0.0,E6 0.0}
DECL BASIS_SUGG_T LAST_BASIS={POINT1[] "P0                      ",POINT2[] "P0                      ",CP_PARAMS[] "CPDAT0                  ",PTP_PARAMS[] "PDAT0                   ",CONT[] "                        ",CP_VEL[] "2                       ",PTP_VEL[] " 100                    ",SYNC_PARAMS[] "SYNCDAT                 ",SPL_NAME[] "S0                      "}
DECL SPOT_SUGG_T LAST_SPOT={GUN[] "1                       ",RETR_CMD[] "#OPN                    ",CHOISE[] "#FIRST                  ",CLO_TM[] "0                       ",PGNO1[] "1                       ",PRESS1[] "0                       ",PGNO2[] "1                       ",PRESS2[] "0                       ",SPOT_PARAMS[] "NORMAL                  "}
DECL E6POS XLO00={X 1447.77295,Y -807.058411,Z 1288.66699,A -0.122811303,B 0.841377616,C -0.772896588,S 2,T 34,E1 0.0,E2 0.0,E3 0.0,E4 0.0,E5 0.0,E6 0.0}
DECL FDAT Flo00={TOOL_NO 1,BASE_NO 2,IPO_FRAME #BASE,POINT2[] " ",TQ_STATE FALSE}
DECL PDAT PPDAT1={VEL 100.0,ACC 100.0,APO_DIST 100.0,APO_MODE #CDIS}
DECL E6POS XLO01={X 1516.36206,Y -814.753296,Z 1289.58398,A -2.64895892,B -2.53534389,C -0.648321629,S 2,T 42,E1 0.0,E2 0.0,E3 0.0,E4 0.0,E5 0.0,E6 0.0}
DECL FDAT Flo01={TOOL_NO 1,BASE_NO 2,IPO_FRAME #BASE,POINT2[] " ",TQ_STATE FALSE}
DECL PDAT PPDAT2={VEL 100.0,ACC 100.0,APO_DIST 100.0,APO_MODE #CDIS}
DECL E6POS XLO03={X 1394.07495,Y 693.451477,Z 1341.46301,A 2.86559391,B 4.28242588,C 0.264305711,S 2,T 43,E1 0.0,E2 0.0,E3 0.0,E4 0.0,E5 0.0,E6 0.0}
DECL FDAT Flo03={TOOL_NO 1,BASE_NO 2,IPO_FRAME #BASE,POINT2[] " ",TQ_STATE FALSE}
DECL PDAT PPDAT4={VEL 100.0,ACC 100.0,APO_DIST 100.0,APO_MODE #CDIS}
DECL E6POS XLO04={X 1522.36304,Y 696.976929,Z 1297.86694,A 3.64751291,B -4.82794523,C -3.60539508,S 2,T 35,E1 0.0,E2 0.0,E3 0.0,E4 0.0,E5 0.0,E6 0.0}
DECL FDAT Flo04={TOOL_NO 1,BASE_NO 2,IPO_FRAME #BASE,POINT2[] " ",TQ_STATE FALSE}
DECL PDAT PPDAT5={VEL 100.0,ACC 100.0,APO_DIST 100.0,APO_MODE #CDIS}
DECL E6POS XLO05={X 1256.854,Y 473.294006,Z 1792.23804,A -113.768997,B -6.72801399,C 11.6442299,S 2,T 3,E1 0.0,E2 0.0,E3 0.0,E4 0.0,E5 0.0,E6 0.0}
DECL FDAT Flo05={TOOL_NO 1,BASE_NO 2,IPO_FRAME #BASE,POINT2[] " ",TQ_STATE FALSE}
DECL PDAT PPDAT6={VEL 100.0,ACC 100.0,APO_DIST 100.0,APO_MODE #CDIS}
DECL LDAT LCPDAT4={VEL 2.0,ACC 100.0,APO_DIST 100.0,APO_FAC 50.0,AXIS_VEL 100.0,AXIS_ACC 100.0,ORI_TYP #VAR,CIRC_TYP #BASE,JERK_FAC 50.0,GEAR_JERK 50.0,EXAX_IGN 0}
DECL E6POS XLO07={X 941.598877,Y -838.958008,Z 1679.10596,A 178.9888,B -7.42855406,C -2.22288799,S 6,T 26,E1 0.0,E2 0.0,E3 0.0,E4 0.0,E5 0.0,E6 0.0}
DECL FDAT Flo07={TOOL_NO 1,BASE_NO 2,IPO_FRAME #BASE,POINT2[] " ",TQ_STATE FALSE}
DECL PDAT PPDAT8={VEL 100.0,ACC 100.0,APO_DIST 100.0,APO_MODE #CDIS}
DECL LDAT LCPDAT6={VEL 2.0,ACC 100.0,APO_DIST 100.0,APO_FAC 50.0,AXIS_VEL 100.0,AXIS_ACC 100.0,ORI_TYP #VAR,CIRC_TYP #BASE,JERK_FAC 50.0,GEAR_JERK 50.0,EXAX_IGN 0}
DECL LDAT LCPDAT11={VEL 2.0,ACC 100.0,APO_DIST 100.0,APO_FAC 50.0,AXIS_VEL 100.0,AXIS_ACC 100.0,ORI_TYP #VAR,CIRC_TYP #BASE,JERK_FAC 50.0,GEAR_JERK 50.0,EXAX_IGN 0}
DECL LDAT LCPDAT12={VEL 2.0,ACC 100.0,APO_DIST 100.0,APO_FAC 50.0,AXIS_VEL 100.0,AXIS_ACC 100.0,ORI_TYP #VAR,CIRC_TYP #BASE,JERK_FAC 50.0,GEAR_JERK 50.0,EXAX_IGN 0}
DECL LDAT LCPDAT13={VEL 2.0,ACC 100.0,APO_DIST 100.0,APO_FAC 50.0,AXIS_VEL 100.0,AXIS_ACC 100.0,ORI_TYP #VAR,CIRC_TYP #BASE,JERK_FAC 50.0,GEAR_JERK 50.0,EXAX_IGN 0}
DECL LDAT LCPDAT14={VEL 2.0,ACC 100.0,APO_DIST 100.0,APO_FAC 50.0,AXIS_VEL 100.0,AXIS_ACC 100.0,ORI_TYP #VAR,CIRC_TYP #BASE,JERK_FAC 50.0,GEAR_JERK 50.0,EXAX_IGN 0}
DECL LDAT LCPDAT15={VEL 2.0,ACC 100.0,APO_DIST 100.0,APO_FAC 50.0,AXIS_VEL 100.0,AXIS_ACC 100.0,ORI_TYP #VAR,CIRC_TYP #BASE,JERK_FAC 50.0,GEAR_JERK 50.0,EXAX_IGN 0}
DECL LDAT LCPDAT16={VEL 2.0,ACC 100.0,APO_DIST 100.0,APO_FAC 50.0,AXIS_VEL 100.0,AXIS_ACC 100.0,ORI_TYP #VAR,CIRC_TYP #BASE,JERK_FAC 50.0,GEAR_JERK 50.0,EXAX_IGN 0}
DECL E6POS XLO16={X 845.884521,Y 696.812378,Z 1404.39502,A 178.004303,B 9.5815258,C -0.273131192,S 6,T 27,E1 0.0,E2 0.0,E3 0.0,E4 0.0,E5 0.0,E6 0.0}
DECL FDAT Flo16={TOOL_NO 1,BASE_NO 2,IPO_FRAME #BASE,POINT2[] " ",TQ_STATE FALSE}
DECL PDAT PPDAT15={VEL 100.0,ACC 100.0,APO_DIST 100.0,APO_MODE #CDIS}
DECL E6POS XLO17={X 784.107727,Y 703.838196,Z 1379.55103,A 173.986298,B 15.6926498,C 4.7314558,S 6,T 27,E1 0.0,E2 0.0,E3 0.0,E4 0.0,E5 0.0,E6 0.0}
DECL FDAT Flo17={TOOL_NO 1,BASE_NO 2,IPO_FRAME #BASE,POINT2[] " ",TQ_STATE FALSE}
DECL E6POS XLO19={X 1124.69604,Y 199.736298,Z 2384.41895,A 149.259796,B 11.4289999,C -5.49499989,S 2,T 35,E1 0.0,E2 0.0,E3 0.0,E4 0.0,E5 0.0,E6 0.0}
DECL FDAT Flo19={TOOL_NO 1,BASE_NO 2,IPO_FRAME #BASE,POINT2[] " ",TQ_STATE FALSE}
DECL PDAT PPDAT17={VEL 100.0,ACC 100.0,APO_DIST 100.0,APO_MODE #CDIS}
DECL E6POS XLO20={X 1281.43604,Y 698.358582,Z 1551.81396,A 2.36923909,B -5.32216883,C -4.31609201,S 2,T 35,E1 0.0,E2 0.0,E3 0.0,E4 0.0,E5 0.0,E6 0.0}
DECL FDAT Flo20={TOOL_NO 1,BASE_NO 2,IPO_FRAME #BASE,POINT2[] " ",TQ_STATE FALSE}
DECL PDAT PPDAT18={VEL 100.0,ACC 100.0,APO_DIST 100.0,APO_MODE #CDIS}
DECL PDAT PPDAT21={VEL 100.0,ACC 100.0,APO_DIST 100.0,APO_MODE #CDIS}
DECL PDAT PPDAT22={VEL 100.0,ACC 100.0,APO_DIST 100.0,APO_MODE #CDIS}
DECL E6POS XLO22={X 900.839294,Y 858.841919,Z 1672.51099,A -166.765305,B 10.6000099,C -6.8331542,S 2,T 11,E1 0.0,E2 0.0,E3 0.0,E4 0.0,E5 0.0,E6 0.0}
DECL FDAT Flo22={TOOL_NO 1,BASE_NO 2,IPO_FRAME #BASE,POINT2[] " ",TQ_STATE FALSE}
DECL PDAT PPDAT25={VEL 100.0,ACC 100.0,APO_DIST 100.0,APO_MODE #CDIS}
DECL PDAT PPDAT27={VEL 100.0,ACC 100.0,APO_DIST 100.0}
DECL E6POS XLO24={X 719.195129,Y 683.543518,Z 1279.51294,A 179.677307,B 6.73365498,C 2.82836199,S 6,T 27,E1 0.0,E2 0.0,E3 0.0,E4 0.0,E5 0.0,E6 0.0}
DECL FDAT Flo24={TOOL_NO 1,BASE_NO 2,IPO_FRAME #BASE,POINT2[] " ",TQ_STATE FALSE}
DECL PDAT PPDAT28={VEL 100.0,ACC 100.0,APO_DIST 100.0,APO_MODE #CDIS}
DECL PDAT PPDAT29={VEL 100.0,ACC 100.0,APO_DIST 100.0}
DECL PDAT PPDAT30={VEL 100.0,ACC 100.0,APO_DIST 100.0,APO_MODE #CDIS}
DECL PDAT PPDAT31={VEL 100.0,ACC 100.0,APO_DIST 100.0,APO_MODE #CDIS}
DECL E6POS XP2={X 1584.198,Y 75.2247696,Z 1334.33997,A 173.334106,B 1.89106405,C -5.68013191,S 2,T 10,E1 0.0,E2 0.0,E3 0.0,E4 0.0,E5 0.0,E6 0.0}
DECL FDAT FP2={TOOL_NO 1,BASE_NO 2,IPO_FRAME #BASE,POINT2[] " ",TQ_STATE FALSE}
DECL PDAT PPDAT33={VEL 100.0,ACC 100.0,APO_DIST 2.0,APO_MODE #CDIS}
DECL E6POS XP3={X -730.218323,Y -2587.86499,Z 4197.75684,A -119.585297,B -72.7684174,C 35.2589111,S 2,T 10,E1 0.0,E2 0.0,E3 0.0,E4 0.0,E5 0.0,E6 0.0}
DECL FDAT FP3={TOOL_NO 1,BASE_NO 2,IPO_FRAME #BASE,POINT2[] " ",TQ_STATE FALSE}
DECL PDAT PPDAT34={VEL 100.0,ACC 100.0,APO_DIST 100.0,APO_MODE #CDIS}
DECL E6POS XP4={X -730.218323,Y -2587.86499,Z 4197.75684,A -119.585297,B -72.7684174,C 35.2589111,S 2,T 10,E1 0.0,E2 0.0,E3 0.0,E4 0.0,E5 0.0,E6 0.0}
DECL FDAT FP4={TOOL_NO 1,BASE_NO 2,IPO_FRAME #BASE,POINT2[] " ",TQ_STATE FALSE}
DECL PDAT PPDAT35={VEL 100.0,ACC 100.0,APO_DIST 100.0,APO_MODE #CDIS}
DECL E6POS XP5={X 1043.37195,Y -820.505005,Z 1455.36304,A -177.823807,B 19.4657803,C 3.59396291,S 2,T 10,E1 0.0,E2 0.0,E3 0.0,E4 0.0,E5 0.0,E6 0.0}
DECL FDAT FP5={TOOL_NO 1,BASE_NO 2,IPO_FRAME #BASE,POINT2[] " ",TQ_STATE FALSE}
DECL PDAT PPDAT36={VEL 100.0,ACC 100.0,APO_DIST 100.0,APO_MODE #CDIS}
DECL E6POS XP6={X 1174.328,Y -1072.65295,Z 1684.19604,A -176.480103,B 14.2246704,C 15.2563295,S 6,T 26,E1 0.0,E2 0.0,E3 0.0,E4 0.0,E5 0.0,E6 0.0}
DECL FDAT FP6={TOOL_NO 1,BASE_NO 2,IPO_FRAME #BASE,POINT2[] " ",TQ_STATE FALSE}
DECL PDAT PPDAT37={VEL 100.0,ACC 100.0,APO_DIST 100.0,APO_MODE #CDIS}
DECL LDAT LCPDAT25={VEL 2.0,ACC 100.0,APO_DIST 100.0,APO_FAC 50.0,AXIS_VEL 100.0,AXIS_ACC 100.0,ORI_TYP #VAR,CIRC_TYP #BASE,JERK_FAC 50.0,GEAR_JERK 50.0,EXAX_IGN 0}
DECL E6POS XP7={X 975.729309,Y -811.65918,Z 1296.86304,A 179.547897,B 19.8234406,C 0.635492921,S 2,T 10,E1 0.0,E2 0.0,E3 0.0,E4 0.0,E5 0.0,E6 0.0}
DECL FDAT FP7={TOOL_NO 1,BASE_NO 2,IPO_FRAME #BASE,POINT2[] " ",TQ_STATE FALSE}
DECL LDAT LCPDAT26={VEL 2.0,ACC 100.0,APO_DIST 100.0,APO_FAC 50.0,AXIS_VEL 100.0,AXIS_ACC 100.0,ORI_TYP #VAR,CIRC_TYP #BASE,JERK_FAC 50.0,GEAR_JERK 50.0,EXAX_IGN 0}
DECL E6POS XP8={X 1043.36597,Y -827.157898,Z 1455.36096,A -177.824005,B 19.4656601,C 3.59387207,S 2,T 10,E1 0.0,E2 0.0,E3 0.0,E4 0.0,E5 0.0,E6 0.0}
DECL FDAT FP8={TOOL_NO 1,BASE_NO 2,IPO_FRAME #BASE,POINT2[] " ",TQ_STATE FALSE}
DECL PDAT PPDAT39={VEL 100.0,ACC 100.0,APO_DIST 100.0}
DECL E6POS XP9={X 1174.328,Y -1072.65295,Z 1684.19604,A -176.480103,B 14.2246704,C 15.2563295,S 6,T 26,E1 0.0,E2 0.0,E3 0.0,E4 0.0,E5 0.0,E6 0.0}
DECL FDAT FP9={TOOL_NO 1,BASE_NO 2,IPO_FRAME #BASE,POINT2[] " ",TQ_STATE FALSE}
DECL PDAT PPDAT40={VEL 100.0,ACC 100.0,APO_DIST 100.0}
ENDDAT
